LIN {X 0,Y 163.128,Z 425.869,A -85,B 0,C 180,E1 -26654.982,E2 -26654.982} C_VEL
LIN {X 0,Y 171.589,Z 416.887,A -85,B 0,C 180,E1 -26656.969,E2 -26656.969} C_VEL
LIN {X 0,Y 179.197,Z 407.097,A -85,B 0,C 180,E1 -26658.583,E2 -26658.583} C_VEL
LIN {X 0,Y 186.048,Z 396.461,A -85,B 0,C 180,E1 -26659.876,E2 -26659.876} C_VEL
LIN {X 0,Y 192.161,Z 384.861,A -85,B 0,C 180,E1 -26660.93,E2 -26660.93} C_VEL
LIN {X 0,Y 196.671,Z 373.993,A -85,B 0,C 180,E1 -26661.72,E2 -26661.72} C_VEL
LIN {X 0,Y 200.139,Z 363.217,A -85,B 0,C 180,E1 -26662.314,E2 -26662.314} C_VEL
LIN {X 0,Y 199.888,Z 363.628,A -85,B 0,C 180,E1 -26665.464,E2 -26665.464} C_VEL
LIN {X 0,Y 199.801,Z 364.596,A -85,B 0,C 180,E1 -26666.634,E2 -26666.634} C_VEL
LIN {X 0,Y 199.425,Z 366.277,A -85,B 0,C 180,E1 -26667.159,E2 -26667.159} C_VEL
LIN {X 0,Y 194.964,Z 379.043,A -85,B 0,C 180,E1 -26667.683,E2 -26667.683} C_VEL
LIN {X 0,Y 188.908,Z 392.245,A -85,B 0,C 180,E1 -26668.498,E2 -26668.498} C_VEL
LIN {X 0,Y 181.772,Z 404.47,A -85,B 0,C 180,E1 -26669.559,E2 -26669.559} C_VEL
LIN {X 0,Y 173.973,Z 415.421,A -85,B 0,C 180,E1 -26670.869,E2 -26670.869} C_VEL
LIN {X 0,Y 164.885,Z 425.886,A -85,B 0,C 180,E1 -26672.677,E2 -26672.677} C_VEL
LIN {X 0,Y 156.103,Z 434.387,A -85,B 0,C 180,E1 -26674.759,E2 -26674.759} C_VEL
LIN {X 0,Y 146.247,Z 442.42,A -85,B 0,C 180,E1 -26677.549,E2 -26677.549} C_VEL
LIN {X 0,Y 138.25,Z 447.941,A -85,B 0,C 180,E1 -26680.319,E2 -26680.319} C_VEL
LIN {X 0,Y 130.692,Z 452.389,A -85,B 0,C 180,E1 -26683.457,E2 -26683.457} C_VEL
LIN {X 0,Y 123.692,Z 455.88,A -85,B 0,C 180,E1 -26687.019,E2 -26687.019} C_VEL
LIN {X 0,Y 115.424,Z 459.143,A -85,B 0,C 180,E1 -26692.495,E2 -26692.495} C_VEL
LIN {X 0,Y 108.504,Z 460.97,A -85,B 0,C 180,E1 -26698.794,E2 -26698.794} C_VEL
LIN {X 0,Y 103.185,Z 461.402,A -85,B 0,C 180,E1 -26705.881,E2 -26705.881} C_VEL
LIN {X 0,Y 99.914,Z 460.389,A -85,B 0,C 180,E1 -26713.66,E2 -26713.66} C_VEL
LIN {X 0,Y 98.634,Z 457.962,A -85,B 0,C 180,E1 -26721.808,E2 -26721.808} C_VEL
LIN {X 0,Y 98.771,Z 454.798,A -85,B 0,C 180,E1 -26728.418,E2 -26728.418} C_VEL
LIN {X 0,Y 98.803,Z 451.965,A -85,B 0,C 180,E1 -26732.782,E2 -26732.782} C_VEL
LIN {X 0,Y 98.851,Z 447.513,A -85,B 0,C 180,E1 -26738.174,E2 -26738.174} C_VEL
LIN {X 0,Y 99.696,Z 441.144,A -85,B 0,C 180,E1 -26744.282,E2 -26744.282} C_VEL
LIN {X 0,Y 101.518,Z 433.131,A -85,B 0,C 180,E1 -26750.249,E2 -26750.249} C_VEL
LIN {X 0,Y 103.699,Z 424.917,A -85,B 0,C 180,E1 -26755.057,E2 -26755.057} C_VEL
LIN {X 0,Y 106.646,Z 414.958,A -85,B 0,C 180,E1 -26759.617,E2 -26759.617} C_VEL
LIN {X 0,Y 109.644,Z 404.598,A -85,B 0,C 180,E1 -26763.239,E2 -26763.239} C_VEL
LIN {X 0,Y 112.675,Z 392.942,A -85,B 0,C 180,E1 -26766.333,E2 -26766.333} C_VEL
LIN {X 0,Y 115.263,Z 381.156,A -85,B 0,C 180,E1 -26768.675,E2 -26768.675} C_VEL
LIN {X 0,Y 117.619,Z 367.853,A -85,B 0,C 180,E1 -26770.521,E2 -26770.521} C_VEL
LIN {X 0,Y 117.914,Z 365.846,A -85,B 0,C 180,E1 -26770.749,E2 -26770.749} C_VEL
LIN {X 0,Y 118.064,Z 360.135,A -85,B 0,C 180,E1 -26771.461,E2 -26771.461} C_VEL
LIN {X 0,Y 116.415,Z 350.753,A -85,B 0,C 180,E1 -26772.801,E2 -26772.801} C_VEL
LIN {X 0,Y 114.613,Z 341.305,A -85,B 0,C 180,E1 -26774.061,E2 -26774.061} C_VEL
LIN {X 0,Y 114.511,Z 335.482,A -85,B 0,C 180,E1 -26774.605,E2 -26774.605} C_VEL
LIN {X 0,Y 115.704,Z 319.854,A -85,B 0,C 180,E1 -26775.743,E2 -26775.743} C_VEL
LIN {X 0,Y 114.812,Z 307.519,A -85,B 0,C 180,E1 -26777.142,E2 -26777.142} C_VEL
LIN {X 0,Y 109.913,Z 291.288,A -85,B 0,C 180,E1 -26780.25,E2 -26780.25} C_VEL
LIN {X 0,Y 105.352,Z 279.17,A -85,B 0,C 180,E1 -26783.198,E2 -26783.198} C_VEL
LIN {X 0,Y 99.994,Z 269.239,A -85,B 0,C 180,E1 -26786.524,E2 -26786.524} C_VEL
LIN {X 0,Y 95.808,Z 262.103,A -85,B 0,C 180,E1 -26789.408,E2 -26789.408} C_VEL
LIN {X 0,Y 94.08,Z 259.671,A -85,B 0,C 180,E1 -26790.642,E2 -26790.642} C_VEL
LIN {X 0,Y 93.573,Z 257.823,A -85,B 0,C 180,E1 -26791.237,E2 -26791.237} C_VEL
LIN {X 0,Y 93.642,Z 257.821,A -85,B 0,C 180,E1 -26797.958,E2 -26797.958} C_VEL
LIN {X 0,Y 94.005,Z 257.76,A -85,B 0,C 180,E1 -26807.038,E2 -26807.038} C_VEL
LIN {X 0,Y 94.117,Z 257.761,A -85,B 0,C 180,E1 -26811.409,E2 -26811.409} C_VEL
LIN {X 0,Y 94.728,Z 257.639,A -85,B 0,C 180,E1 -26819.998,E2 -26819.998} C_VEL
LIN {X 0,Y 94.142,Z 257.758,A -85,B 0,C 180,E1 -26828.585,E2 -26828.585} C_VEL
LIN {X 0,Y 93.991,Z 257.751,A -85,B 0,C 180,E1 -26833.606,E2 -26833.606} C_VEL
LIN {X 0,Y 93.679,Z 257.773,A -85,B 0,C 180,E1 -26842.03,E2 -26842.03} C_VEL
LIN {X 0,Y 93.611,Z 257.818,A -85,B 0,C 180,E1 -26846.772,E2 -26846.772} C_VEL
LIN {X 0,Y 93.588,Z 257.807,A -85,B 0,C 180,E1 -26854.316,E2 -26854.316} C_VEL
LIN {X 0,Y 93.537,Z 257.792,A -85,B 0,C 180,E1 -26862.547,E2 -26862.547} C_VEL
LIN {X 0,Y 93.53,Z 257.835,A -85,B 0,C 180,E1 -26868.711,E2 -26868.711} C_VEL
LIN {X 0,Y 93.579,Z 257.793,A -85,B 0,C 180,E1 -26875.7,E2 -26875.7} C_VEL
LIN {X 0,Y 93.664,Z 257.819,A -85,B 0,C 180,E1 -26884.209,E2 -26884.209} C_VEL
LIN {X 0,Y 93.691,Z 257.806,A -85,B 0,C 180,E1 -26887.975,E2 -26887.975} C_VEL
LIN {X 0,Y 94.089,Z 257.765,A -85,B 0,C 180,E1 -26897.053,E2 -26897.053} C_VEL
LIN {X 0,Y 94.12,Z 257.747,A -85,B 0,C 180,E1 -26900.058,E2 -26900.058} C_VEL
LIN {X 0,Y 95.242,Z 260.722,A -85,B 0,C 180,E1 -26901.106,E2 -26901.106} C_VEL
LIN {X 0,Y 96.858,Z 262.736,A -85,B 0,C 180,E1 -26902.193,E2 -26902.193} C_VEL
LIN {X 0,Y 98.996,Z 266.163,A -85,B 0,C 180,E1 -26903.652,E2 -26903.652} C_VEL
LIN {X 0,Y 102.442,Z 271.693,A -85,B 0,C 180,E1 -26905.821,E2 -26905.821} C_VEL
LIN {X 0,Y 109.777,Z 287.544,A -85,B 0,C 180,E1 -26910.3,E2 -26910.3} C_VEL
LIN {X 0,Y 116.248,Z 304.133,A -85,B 0,C 180,E1 -26913.943,E2 -26913.943} C_VEL
LIN {X 0,Y 116.608,Z 305.841,A -85,B 0,C 180,E1 -26914.203,E2 -26914.203} C_VEL
LIN {X 0,Y 112.302,Z 350.785,A -85,B 0,C 180,E1 -26917.359,E2 -26917.359} C_VEL
LIN {X 0,Y 110.494,Z 363.82,A -85,B 0,C 180,E1 -26918.918,E2 -26918.918} C_VEL
LIN {X 0,Y 107.94,Z 377.265,A -85,B 0,C 180,E1 -26921.263,E2 -26921.263} C_VEL
LIN {X 0,Y 104.836,Z 389.887,A -85,B 0,C 180,E1 -26924.32,E2 -26924.32} C_VEL
LIN {X 0,Y 101.801,Z 401.041,A -85,B 0,C 180,E1 -26927.94,E2 -26927.94} C_VEL
LIN {X 0,Y 98.733,Z 411.262,A -85,B 0,C 180,E1 -26932.281,E2 -26932.281} C_VEL
LIN {X 0,Y 96.103,Z 419.877,A -85,B 0,C 180,E1 -26936.942,E2 -26936.942} C_VEL
LIN {X 0,Y 93.655,Z 428.33,A -85,B 0,C 180,E1 -26942.751,E2 -26942.751} C_VEL
LIN {X 0,Y 92.06,Z 435.208,A -85,B 0,C 180,E1 -26948.791,E2 -26948.791} C_VEL
LIN {X 0,Y 90.924,Z 441.541,A -85,B 0,C 180,E1 -26955.923,E2 -26955.923} C_VEL
LIN {X 0,Y 90.75,Z 445.601,A -85,B 0,C 180,E1 -26961.719,E2 -26961.719} C_VEL
LIN {X 0,Y 91.999,Z 450.233,A -85,B 0,C 180,E1 -26970.372,E2 -26970.372} C_VEL
LIN {X 0,Y 94.797,Z 453.146,A -85,B 0,C 180,E1 -26978.244,E2 -26978.244} C_VEL
LIN {X 0,Y 97.638,Z 454.379,A -85,B 0,C 180,E1 -26983.268,E2 -26983.268} C_VEL
LIN {X 0,Y 101.113,Z 454.988,A -85,B 0,C 180,E1 -26987.966,E2 -26987.966} C_VEL
LIN {X 0,Y 106.154,Z 454.979,A -85,B 0,C 180,E1 -26993.205,E2 -26993.205} C_VEL
LIN {X 0,Y 112.489,Z 454.028,A -85,B 0,C 180,E1 -26998.241,E2 -26998.241} C_VEL
LIN {X 0,Y 120.795,Z 451.707,A -85,B 0,C 180,E1 -27003.337,E2 -27003.337} C_VEL
LIN {X 0,Y 130.29,Z 447.868,A -85,B 0,C 180,E1 -27007.85,E2 -27007.85} C_VEL
LIN {X 0,Y 140.094,Z 442.584,A -85,B 0,C 180,E1 -27011.577,E2 -27011.577} C_VEL
LIN {X 0,Y 148.86,Z 436.826,A -85,B 0,C 180,E1 -27014.291,E2 -27014.291} C_VEL
LIN {X 0,Y 158.415,Z 429.249,A -85,B 0,C 180,E1 -27016.761,E2 -27016.761} C_VEL
LIN {X 0,Y 167.121,Z 420.854,A -85,B 0,C 180,E1 -27018.71,E2 -27018.71} C_VEL
LIN {X 0,Y 175.528,Z 411.15,A -85,B 0,C 180,E1 -27020.387,E2 -27020.387} C_VEL
LIN {X 0,Y 183.337,Z 400.242,A -85,B 0,C 180,E1 -27021.732,E2 -27021.732} C_VEL
LIN {X 0,Y 189.266,Z 390.03,A -85,B 0,C 180,E1 -27022.696,E2 -27022.696} C_VEL
LIN {X 0,Y 195.03,Z 377.557,A -85,B 0,C 180,E1 -27023.606,E2 -27023.606} C_VEL
LIN {X 0,Y 197.721,Z 370.368,A -85,B 0,C 180,E1 -27024.018,E2 -27024.018} C_VEL
LIN {X 0,Y 197.801,Z 370.092,A -85,B 0,C 180,E1 -27024.219,E2 -27024.219} C_VEL
LIN {X 0,Y 197.787,Z 370.277,A -85,B 0,C 180,E1 -27025.066,E2 -27025.066} C_VEL
LIN {X 0,Y 197.46,Z 371.297,A -85,B 0,C 180,E1 -27025.267,E2 -27025.267} C_VEL
LIN {X 0,Y 192.672,Z 383.338,A -85,B 0,C 180,E1 -27025.795,E2 -27025.795} C_VEL
LIN {X 0,Y 186.571,Z 395.367,A -85,B 0,C 180,E1 -27026.549,E2 -27026.549} C_VEL
LIN {X 0,Y 179.278,Z 406.879,A -85,B 0,C 180,E1 -27027.521,E2 -27027.521} C_VEL
LIN {X 0,Y 172.115,Z 416.231,A -85,B 0,C 180,E1 -27028.62,E2 -27028.62} C_VEL
LIN {X 0,Y 162.783,Z 426.49,A -85,B 0,C 180,E1 -27030.301,E2 -27030.301} C_VEL
LIN {X 0,Y 153.733,Z 434.831,A -85,B 0,C 180,E1 -27032.259,E2 -27032.259} C_VEL
LIN {X 0,Y 144.941,Z 441.634,A -85,B 0,C 180,E1 -27034.491,E2 -27034.491} C_VEL
LIN {X 0,Y 133.814,Z 448.805,A -85,B 0,C 180,E1 -27038.026,E2 -27038.026} C_VEL
LIN {X 0,Y 125.938,Z 452.982,A -85,B 0,C 180,E1 -27041.124,E2 -27041.124} C_VEL
LIN {X 0,Y 118.613,Z 456.212,A -85,B 0,C 180,E1 -27044.688,E2 -27044.688} C_VEL
LIN {X 0,Y 109.877,Z 459.205,A -85,B 0,C 180,E1 -27050.241,E2 -27050.241} C_VEL
LIN {X 0,Y 102.489,Z 460.771,A -85,B 0,C 180,E1 -27056.734,E2 -27056.734} C_VEL
LIN {X 0,Y 96.746,Z 460.91,A -85,B 0,C 180,E1 -27064.162,E2 -27064.162} C_VEL
LIN {X 0,Y 93.117,Z 459.687,A -85,B 0,C 180,E1 -27072.43,E2 -27072.43} C_VEL
LIN {X 0,Y 91.655,Z 457.019,A -85,B 0,C 180,E1 -27081.179,E2 -27081.179} C_VEL
LIN {X 0,Y 91.753,Z 453.772,A -85,B 0,C 180,E1 -27088.145,E2 -27088.145} C_VEL
LIN {X 0,Y 91.795,Z 450.795,A -85,B 0,C 180,E1 -27092.821,E2 -27092.821} C_VEL
LIN {X 0,Y 91.961,Z 444.993,A -85,B 0,C 180,E1 -27099.9,E2 -27099.9} C_VEL
LIN {X 0,Y 93.125,Z 438.095,A -85,B 0,C 180,E1 -27106.438,E2 -27106.438} C_VEL
LIN {X 0,Y 95.385,Z 429.412,A -85,B 0,C 180,E1 -27112.754,E2 -27112.754} C_VEL
LIN {X 0,Y 97.953,Z 420.469,A -85,B 0,C 180,E1 -27117.795,E2 -27117.795} C_VEL
LIN {X 0,Y 100.887,Z 410.694,A -85,B 0,C 180,E1 -27122.08,E2 -27122.08} C_VEL
LIN {X 0,Y 104.043,Z 399.823,A -85,B 0,C 180,E1 -27125.71,E2 -27125.71} C_VEL
LIN {X 0,Y 107.046,Z 388.339,A -85,B 0,C 180,E1 -27128.582,E2 -27128.582} C_VEL
LIN {X 0,Y 109.87,Z 375.3,A -85,B 0,C 180,E1 -27130.963,E2 -27130.963} C_VEL
LIN {X 0,Y 112.097,Z 361.245,A -85,B 0,C 180,E1 -27132.673,E2 -27132.673} C_VEL
LIN {X 0,Y 114.511,Z 335.482,A -85,B 0,C 180,E1 -27134.605,E2 -27134.605} C_VEL
LIN {X 0,Y 114.425,Z 329.67,A -85,B 0,C 180,E1 -27135.168,E2 -27135.168} C_VEL
LIN {X 0,Y 113.409,Z 324.025,A -85,B 0,C 180,E1 -27135.972,E2 -27135.972} C_VEL
LIN {X 0,Y 107.787,Z 305.825,A -85,B 0,C 180,E1 -27139.468,E2 -27139.468} C_VEL
LIN {X 0,Y 102.649,Z 289.521,A -85,B 0,C 180,E1 -27143.091,E2 -27143.091} C_VEL
LIN {X 0,Y 99.916,Z 282.46,A -85,B 0,C 180,E1 -27144.99,E2 -27144.99} C_VEL
LIN {X 0,Y 94.449,Z 272.371,A -85,B 0,C 180,E1 -27148.763,E2 -27148.763} C_VEL
LIN {X 0,Y 91.1,Z 266.722,A -85,B 0,C 180,E1 -27151.329,E2 -27151.329} C_VEL
LIN {X 0,Y 88.937,Z 263.157,A -85,B 0,C 180,E1 -27153.096,E2 -27153.096} C_VEL
LIN {X 0,Y 87.203,Z 260.823,A -85,B 0,C 180,E1 -27154.514,E2 -27154.514} C_VEL
LIN {X 0,Y 86.551,Z 258.691,A -85,B 0,C 180,E1 -27155.324,E2 -27155.324} C_VEL
LIN {X 0,Y 86.586,Z 258.685,A -85,B 0,C 180,E1 -27161.053,E2 -27161.053} C_VEL
LIN {X 0,Y 86.848,Z 258.643,A -85,B 0,C 180,E1 -27166.157,E2 -27166.157} C_VEL
LIN {X 0,Y 87.012,Z 258.647,A -85,B 0,C 180,E1 -27170.702,E2 -27170.702} C_VEL
LIN {X 0,Y 87.66,Z 258.517,A -85,B 0,C 180,E1 -27179.998,E2 -27179.998} C_VEL
LIN {X 0,Y 87.052,Z 258.64,A -85,B 0,C 180,E1 -27189.29,E2 -27189.29} C_VEL
LIN {X 0,Y 86.884,Z 258.629,A -85,B 0,C 180,E1 -27194.042,E2 -27194.042} C_VEL
LIN {X 0,Y 86.617,Z 258.63,A -85,B 0,C 180,E1 -27198.937,E2 -27198.937} C_VEL
LIN {X 0,Y 86.574,Z 258.695,A -85,B 0,C 180,E1 -27206.764,E2 -27206.764} C_VEL
LIN {X 0,Y 86.509,Z 258.673,A -85,B 0,C 180,E1 -27215.679,E2 -27215.679} C_VEL
LIN {X 0,Y 86.478,Z 258.673,A -85,B 0,C 180,E1 -27223.001,E2 -27223.001} C_VEL
LIN {X 0,Y 86.451,Z 258.717,A -85,B 0,C 180,E1 -27229.437,E2 -27229.437} C_VEL
LIN {X 0,Y 86.522,Z 258.673,A -85,B 0,C 180,E1 -27235.353,E2 -27235.353} C_VEL
LIN {X 0,Y 86.578,Z 258.697,A -85,B 0,C 180,E1 -27243.24,E2 -27243.24} C_VEL
LIN {X 0,Y 86.645,Z 258.667,A -85,B 0,C 180,E1 -27251.07,E2 -27251.07} C_VEL
LIN {X 0,Y 86.973,Z 258.822,A -85,B 0,C 180,E1 -27256.047,E2 -27256.047} C_VEL
LIN {X 0,Y 88.098,Z 261.576,A -85,B 0,C 180,E1 -27257.182,E2 -27257.182} C_VEL
LIN {X 0,Y 89.958,Z 263.827,A -85,B 0,C 180,E1 -27258.627,E2 -27258.627} C_VEL
LIN {X 0,Y 92.146,Z 267.211,A -85,B 0,C 180,E1 -27260.313,E2 -27260.313} C_VEL
LIN {X 0,Y 97.679,Z 276.274,A -85,B 0,C 180,E1 -27264.283,E2 -27264.283} C_VEL
LIN {X 0,Y 104.482,Z 291.419,A -85,B 0,C 180,E1 -27268.816,E2 -27268.816} C_VEL
LIN {X 0,Y 110.395,Z 306.934,A -85,B 0,C 180,E1 -27272.467,E2 -27272.467} C_VEL
LIN {X 0,Y 105.939,Z 351.171,A -85,B 0,C 180,E1 -27275.689,E2 -27275.689} C_VEL
LIN {X 0,Y 103.843,Z 365.269,A -85,B 0,C 180,E1 -27277.473,E2 -27277.473} C_VEL
LIN {X 0,Y 101.404,Z 377.429,A -85,B 0,C 180,E1 -27279.725,E2 -27279.725} C_VEL
LIN {X 0,Y 98.186,Z 390.026,A -85,B 0,C 180,E1 -27282.924,E2 -27282.924} C_VEL
LIN {X 0,Y 95.015,Z 401.091,A -85,B 0,C 180,E1 -27286.703,E2 -27286.703} C_VEL
LIN {X 0,Y 91.908,Z 410.953,A -85,B 0,C 180,E1 -27291.129,E2 -27291.129} C_VEL
LIN {X 0,Y 88.674,Z 421.047,A -85,B 0,C 180,E1 -27297.051,E2 -27297.051} C_VEL
LIN {X 0,Y 86.255,Z 429.325,A -85,B 0,C 180,E1 -27303.362,E2 -27303.362} C_VEL
LIN {X 0,Y 84.686,Z 436.002,A -85,B 0,C 180,E1 -27309.859,E2 -27309.859} C_VEL
LIN {X 0,Y 83.83,Z 441.309,A -85,B 0,C 180,E1 -27316.333,E2 -27316.333} C_VEL
LIN {X 0,Y 83.824,Z 446.332,A -85,B 0,C 180,E1 -27324.065,E2 -27324.065} C_VEL
LIN {X 0,Y 84.793,Z 449.444,A -85,B 0,C 180,E1 -27330.18,E2 -27330.18} C_VEL
LIN {X 0,Y 86.531,Z 451.862,A -85,B 0,C 180,E1 -27336.042,E2 -27336.042} C_VEL
LIN {X 0,Y 89.077,Z 453.627,A -85,B 0,C 180,E1 -27341.605,E2 -27341.605} C_VEL
LIN {X 0,Y 93.365,Z 455.008,A -85,B 0,C 180,E1 -27348.087,E2 -27348.087} C_VEL
LIN {X 0,Y 98.901,Z 455.475,A -85,B 0,C 180,E1 -27354.124,E2 -27354.124} C_VEL
LIN {X 0,Y 106.196,Z 454.869,A -85,B 0,C 180,E1 -27360.001,E2 -27360.001} C_VEL
LIN {X 0,Y 112.72,Z 453.53,A -85,B 0,C 180,E1 -27364.071,E2 -27364.071} C_VEL
LIN {X 0,Y 120.648,Z 451.105,A -85,B 0,C 180,E1 -27368.035,E2 -27368.035} C_VEL
LIN {X 0,Y 131.42,Z 446.582,A -85,B 0,C 180,E1 -27372.353,E2 -27372.353} C_VEL
LIN {X 0,Y 142.298,Z 440.543,A -85,B 0,C 180,E1 -27375.763,E2 -27375.763} C_VEL
LIN {X 0,Y 152.107,Z 433.74,A -85,B 0,C 180,E1 -27378.255,E2 -27378.255} C_VEL
LIN {X 0,Y 161.786,Z 425.663,A -85,B 0,C 180,E1 -27380.337,E2 -27380.337} C_VEL
LIN {X 0,Y 169.833,Z 417.552,A -85,B 0,C 180,E1 -27381.867,E2 -27381.867} C_VEL
LIN {X 0,Y 178.101,Z 407.515,A -85,B 0,C 180,E1 -27383.242,E2 -27383.242} C_VEL
LIN {X 0,Y 185.063,Z 397.262,A -85,B 0,C 180,E1 -27384.31,E2 -27384.31} C_VEL
LIN {X 0,Y 185.261,Z 396.969,A -85,B 0,C 180,E1 -27384.446,E2 -27384.446} C_VEL
LIN {X 0,Y 177.848,Z 408.08,A -85,B 0,C 180,E1 -27385.331,E2 -27385.331} C_VEL
LIN {X 0,Y 168.922,Z 419.053,A -85,B 0,C 180,E1 -27386.567,E2 -27386.567} C_VEL
LIN {X 0,Y 159.408,Z 428.609,A -85,B 0,C 180,E1 -27388.156,E2 -27388.156} C_VEL
LIN {X 0,Y 148.607,Z 437.623,A -85,B 0,C 180,E1 -27390.346,E2 -27390.346} C_VEL
LIN {X 0,Y 138.166,Z 444.759,A -85,B 0,C 180,E1 -27392.943,E2 -27392.943} C_VEL
LIN {X 0,Y 126.82,Z 451.066,A -85,B 0,C 180,E1 -27396.538,E2 -27396.538} C_VEL
LIN {X 0,Y 118.792,Z 454.631,A -85,B 0,C 180,E1 -27399.733,E2 -27399.733} C_VEL
LIN {X 0,Y 113.743,Z 456.55,A -85,B 0,C 180,E1 -27402.151,E2 -27402.151} C_VEL
LIN {X 0,Y 104.505,Z 459.218,A -85,B 0,C 180,E1 -27407.745,E2 -27407.745} C_VEL
LIN {X 0,Y 96.625,Z 460.493,A -85,B 0,C 180,E1 -27414.421,E2 -27414.421} C_VEL
LIN {X 0,Y 90.41,Z 460.407,A -85,B 0,C 180,E1 -27422.202,E2 -27422.202} C_VEL
LIN {X 0,Y 86.376,Z 458.929,A -85,B 0,C 180,E1 -27431.008,E2 -27431.008} C_VEL
LIN {X 0,Y 84.713,Z 455.996,A -85,B 0,C 180,E1 -27440.45,E2 -27440.45} C_VEL
LIN {X 0,Y 84.781,Z 452.603,A -85,B 0,C 180,E1 -27447.86,E2 -27447.86} C_VEL
LIN {X 0,Y 84.776,Z 449.419,A -85,B 0,C 180,E1 -27453.064,E2 -27453.064} C_VEL
LIN {X 0,Y 85.021,Z 443.356,A -85,B 0,C 180,E1 -27460.717,E2 -27460.717} C_VEL
LIN {X 0,Y 86.343,Z 436.124,A -85,B 0,C 180,E1 -27467.77,E2 -27467.77} C_VEL
LIN {X 0,Y 88.843,Z 427.113,A -85,B 0,C 180,E1 -27474.535,E2 -27474.535} C_VEL
LIN {X 0,Y 92.092,Z 416.683,A -85,B 0,C 180,E1 -27480.366,E2 -27480.366} C_VEL
LIN {X 0,Y 95.395,Z 406.131,A -85,B 0,C 180,E1 -27484.812,E2 -27484.812} C_VEL
LIN {X 0,Y 98.895,Z 394.05,A -85,B 0,C 180,E1 -27488.58,E2 -27488.58} C_VEL
LIN {X 0,Y 102.108,Z 381.146,A -85,B 0,C 180,E1 -27491.483,E2 -27491.483} C_VEL
LIN {X 0,Y 104.615,Z 368.197,A -85,B 0,C 180,E1 -27493.512,E2 -27493.512} C_VEL
LIN {X 0,Y 106.437,Z 354.841,A -85,B 0,C 180,E1 -27494.879,E2 -27494.879} C_VEL
LIN {X 0,Y 109.49,Z 320.718,A -85,B 0,C 180,E1 -27497.421,E2 -27497.421} C_VEL
LIN {X 0,Y 108.795,Z 309.728,A -85,B 0,C 180,E1 -27498.742,E2 -27498.742} C_VEL
LIN {X 0,Y 107.787,Z 305.825,A -85,B 0,C 180,E1 -27499.468,E2 -27499.468} C_VEL
LIN {X 0,Y 105.834,Z 300.741,A -85,B 0,C 180,E1 -27500.676,E2 -27500.676} C_VEL
LIN {X 0,Y 103.066,Z 296.263,A -85,B 0,C 180,E1 -27502.188,E2 -27502.188} C_VEL
LIN {X 0,Y 94.591,Z 285.371,A -85,B 0,C 180,E1 -27507.016,E2 -27507.016} C_VEL
LIN {X 0,Y 92.822,Z 282.379,A -85,B 0,C 180,E1 -27508.273,E2 -27508.273} C_VEL
LIN {X 0,Y 87.205,Z 272.194,A -85,B 0,C 180,E1 -27512.811,E2 -27512.811} C_VEL
LIN {X 0,Y 84.154,Z 267.566,A -85,B 0,C 180,E1 -27515.482,E2 -27515.482} C_VEL
LIN {X 0,Y 82.237,Z 264.377,A -85,B 0,C 180,E1 -27517.381,E2 -27517.381} C_VEL
LIN {X 0,Y 80.259,Z 262.081,A -85,B 0,C 180,E1 -27519.327,E2 -27519.327} C_VEL
LIN {X 0,Y 79.527,Z 259.567,A -85,B 0,C 180,E1 -27520.644,E2 -27520.644} C_VEL
LIN {X 0,Y 79.765,Z 259.521,A -85,B 0,C 180,E1 -27525.716,E2 -27525.716} C_VEL
LIN {X 0,Y 79.897,Z 259.532,A -85,B 0,C 180,E1 -27529.866,E2 -27529.866} C_VEL
LIN {X 0,Y 80.591,Z 259.396,A -85,B 0,C 180,E1 -27539.998,E2 -27539.998} C_VEL
LIN {X 0,Y 79.935,Z 259.523,A -85,B 0,C 180,E1 -27550.126,E2 -27550.126} C_VEL
LIN {X 0,Y 79.717,Z 259.504,A -85,B 0,C 180,E1 -27555.335,E2 -27555.335} C_VEL
LIN {X 0,Y 79.492,Z 259.522,A -85,B 0,C 180,E1 -27560.708,E2 -27560.708} C_VEL
LIN {X 0,Y 79.472,Z 259.583,A -85,B 0,C 180,E1 -27567.843,E2 -27567.843} C_VEL
LIN {X 0,Y 79.374,Z 259.59,A -85,B 0,C 180,E1 -27572.088,E2 -27572.088} C_VEL
LIN {X 0,Y 79.367,Z 259.539,A -85,B 0,C 180,E1 -27578.303,E2 -27578.303} C_VEL
LIN {X 0,Y 79.404,Z 259.574,A -85,B 0,C 180,E1 -27585.076,E2 -27585.076} C_VEL
LIN {X 0,Y 79.379,Z 259.583,A -85,B 0,C 180,E1 -27592.826,E2 -27592.826} C_VEL
LIN {X 0,Y 79.369,Z 259.555,A -85,B 0,C 180,E1 -27597.912,E2 -27597.912} C_VEL
LIN {X 0,Y 79.52,Z 259.578,A -85,B 0,C 180,E1 -27603.778,E2 -27603.778} C_VEL
LIN {X 0,Y 79.599,Z 259.729,A -85,B 0,C 180,E1 -27610.689,E2 -27610.689} C_VEL
LIN {X 0,Y 80.704,Z 262.533,A -85,B 0,C 180,E1 -27612.086,E2 -27612.086} C_VEL
LIN {X 0,Y 83.202,Z 265.112,A -85,B 0,C 180,E1 -27614.446,E2 -27614.446} C_VEL
LIN {X 0,Y 85.468,Z 268.513,A -85,B 0,C 180,E1 -27616.553,E2 -27616.553} C_VEL
LIN {X 0,Y 92.73,Z 280.259,A -85,B 0,C 180,E1 -27622.378,E2 -27622.378} C_VEL
LIN {X 0,Y 99.152,Z 295.087,A -85,B 0,C 180,E1 -27627.175,E2 -27627.175} C_VEL
LIN {X 0,Y 104.228,Z 308.469,A -85,B 0,C 180,E1 -27630.562,E2 -27630.562} C_VEL
LIN {X 0,Y 99.648,Z 351.758,A -85,B 0,C 180,E1 -27633.872,E2 -27633.872} C_VEL
LIN {X 0,Y 97.425,Z 365.715,A -85,B 0,C 180,E1 -27635.724,E2 -27635.724} C_VEL
LIN {X 0,Y 94.642,Z 378.579,A -85,B 0,C 180,E1 -27638.265,E2 -27638.265} C_VEL
LIN {X 0,Y 91.285,Z 390.948,A -85,B 0,C 180,E1 -27641.643,E2 -27641.643} C_VEL
LIN {X 0,Y 87.982,Z 401.823,A -85,B 0,C 180,E1 -27645.659,E2 -27645.659} C_VEL
LIN {X 0,Y 84.548,Z 412.241,A -85,B 0,C 180,E1 -27650.772,E2 -27650.772} C_VEL
LIN {X 0,Y 81.217,Z 422.183,A -85,B 0,C 180,E1 -27657.203,E2 -27657.203} C_VEL
LIN {X 0,Y 78.835,Z 430.291,A -85,B 0,C 180,E1 -27664.102,E2 -27664.102} C_VEL
LIN {X 0,Y 77.322,Z 436.817,A -85,B 0,C 180,E1 -27671.192,E2 -27671.192} C_VEL
LIN {X 0,Y 76.7,Z 441.235,A -85,B 0,C 180,E1 -27677.135,E2 -27677.135} C_VEL
LIN {X 0,Y 77.034,Z 446.961,A -85,B 0,C 180,E1 -27686.814,E2 -27686.814} C_VEL
LIN {X 0,Y 79.458,Z 451.306,A -85,B 0,C 180,E1 -27696.643,E2 -27696.643} C_VEL
LIN {X 0,Y 83.696,Z 454.109,A -85,B 0,C 180,E1 -27705.411,E2 -27705.411} C_VEL
LIN {X 0,Y 87.555,Z 455.237,A -85,B 0,C 180,E1 -27710.764,E2 -27710.764} C_VEL
LIN {X 0,Y 92.091,Z 455.805,A -85,B 0,C 180,E1 -27715.625,E2 -27715.625} C_VEL
LIN {X 0,Y 98.393,Z 455.724,A -85,B 0,C 180,E1 -27720.863,E2 -27720.863} C_VEL
LIN {X 0,Y 105.926,Z 454.727,A -85,B 0,C 180,E1 -27725.662,E2 -27725.662} C_VEL
LIN {X 0,Y 115.801,Z 452.303,A -85,B 0,C 180,E1 -27730.492,E2 -27730.492} C_VEL
LIN {X 0,Y 126.301,Z 448.477,A -85,B 0,C 180,E1 -27734.502,E2 -27734.502} C_VEL
LIN {X 0,Y 137.563,Z 442.928,A -85,B 0,C 180,E1 -27737.852,E2 -27737.852} C_VEL
LIN {X 0,Y 148.333,Z 436.272,A -85,B 0,C 180,E1 -27740.43,E2 -27740.43} C_VEL
LIN {X 0,Y 157.231,Z 429.516,A -85,B 0,C 180,E1 -27742.226,E2 -27742.226} C_VEL
LIN {X 0,Y 166.373,Z 421.141,A -85,B 0,C 180,E1 -27743.833,E2 -27743.833} C_VEL
LIN {X 0,Y 165.956,Z 421.632,A -85,B 0,C 180,E1 -27744.44,E2 -27744.44} C_VEL
LIN {X 0,Y 156.256,Z 430.695,A -85,B 0,C 180,E1 -27745.914,E2 -27745.914} C_VEL
LIN {X 0,Y 145.209,Z 439.14,A -85,B 0,C 180,E1 -27747.97,E2 -27747.97} C_VEL
LIN {X 0,Y 134.478,Z 445.863,A -85,B 0,C 180,E1 -27750.433,E2 -27750.433} C_VEL
LIN {X 0,Y 125.62,Z 450.454,A -85,B 0,C 180,E1 -27752.954,E2 -27752.954} C_VEL
LIN {X 0,Y 117.126,Z 454.063,A -85,B 0,C 180,E1 -27755.908,E2 -27755.908} C_VEL
LIN {X 0,Y 109.104,Z 456.792,A -85,B 0,C 180,E1 -27759.384,E2 -27759.384} C_VEL
LIN {X 0,Y 98.991,Z 459.262,A -85,B 0,C 180,E1 -27765.234,E2 -27765.234} C_VEL
LIN {X 0,Y 90.94,Z 460.209,A -85,B 0,C 180,E1 -27771.816,E2 -27771.816} C_VEL
LIN {X 0,Y 84.199,Z 459.826,A -85,B 0,C 180,E1 -27779.949,E2 -27779.949} C_VEL
LIN {X 0,Y 79.72,Z 458.085,A -85,B 0,C 180,E1 -27789.353,E2 -27789.353} C_VEL
LIN {X 0,Y 77.784,Z 454.951,A -85,B 0,C 180,E1 -27799.59,E2 -27799.59} C_VEL
LIN {X 0,Y 77.784,Z 451.568,A -85,B 0,C 180,E1 -27807.245,E2 -27807.245} C_VEL
LIN {X 0,Y 77.779,Z 449.051,A -85,B 0,C 180,E1 -27811.664,E2 -27811.664} C_VEL
LIN {X 0,Y 77.845,Z 443.86,A -85,B 0,C 180,E1 -27818.958,E2 -27818.958} C_VEL
LIN {X 0,Y 79.019,Z 436.749,A -85,B 0,C 180,E1 -27826.799,E2 -27826.799} C_VEL
LIN {X 0,Y 81.474,Z 427.975,A -85,B 0,C 180,E1 -27834.185,E2 -27834.185} C_VEL
LIN {X 0,Y 84.302,Z 418.926,A -85,B 0,C 180,E1 -27840.009,E2 -27840.009} C_VEL
LIN {X 0,Y 87.571,Z 408.991,A -85,B 0,C 180,E1 -27844.872,E2 -27844.872} C_VEL
LIN {X 0,Y 90.915,Z 398.496,A -85,B 0,C 180,E1 -27848.734,E2 -27848.734} C_VEL
LIN {X 0,Y 94.39,Z 386.225,A -85,B 0,C 180,E1 -27852.07,E2 -27852.07} C_VEL
LIN {X 0,Y 97.217,Z 373.942,A -85,B 0,C 180,E1 -27854.446,E2 -27854.446} C_VEL
LIN {X 0,Y 99.62,Z 359.76,A -85,B 0,C 180,E1 -27856.279,E2 -27856.279} C_VEL
LIN {X 0,Y 103.367,Z 321.146,A -85,B 0,C 180,E1 -27859.351,E2 -27859.351} C_VEL
LIN {X 0,Y 102.852,Z 311.765,A -85,B 0,C 180,E1 -27860.554,E2 -27860.554} C_VEL
LIN {X 0,Y 98.473,Z 296.576,A -85,B 0,C 180,E1 -27863.926,E2 -27863.926} C_VEL
LIN {X 0,Y 94.877,Z 286.554,A -85,B 0,C 180,E1 -27866.726,E2 -27866.726} C_VEL
LIN {X 0,Y 92.822,Z 282.379,A -85,B 0,C 180,E1 -27868.273,E2 -27868.273} C_VEL
LIN {X 0,Y 90.834,Z 279.827,A -85,B 0,C 180,E1 -27869.672,E2 -27869.672} C_VEL
LIN {X 0,Y 86.531,Z 277.148,A -85,B 0,C 180,E1 -27872.484,E2 -27872.484} C_VEL
LIN {X 0,Y 82.202,Z 274.75,A -85,B 0,C 180,E1 -27875.68,E2 -27875.68} C_VEL
LIN {X 0,Y 80.113,Z 272.58,A -85,B 0,C 180,E1 -27877.589,E2 -27877.589} C_VEL
LIN {X 0,Y 78.377,Z 269.787,A -85,B 0,C 180,E1 -27879.494,E2 -27879.494} C_VEL
LIN {X 0,Y 76.283,Z 266.816,A -85,B 0,C 180,E1 -27881.882,E2 -27881.882} C_VEL
LIN {X 0,Y 75.485,Z 265.352,A -85,B 0,C 180,E1 -27882.909,E2 -27882.909} C_VEL
LIN {X 0,Y 73.572,Z 263.048,A -85,B 0,C 180,E1 -27885.299,E2 -27885.299} C_VEL
LIN {X 0,Y 72.734,Z 260.403,A -85,B 0,C 180,E1 -27886.909,E2 -27886.909} C_VEL
LIN {X 0,Y 72.967,Z 260.374,A -85,B 0,C 180,E1 -27894.471,E2 -27894.471} C_VEL
LIN {X 0,Y 73.521,Z 260.275,A -85,B 0,C 180,E1 -27899.998,E2 -27899.998} C_VEL
LIN {X 0,Y 72.829,Z 260.402,A -85,B 0,C 180,E1 -27911.126,E2 -27911.126} C_VEL
LIN {X 0,Y 72.553,Z 260.382,A -85,B 0,C 180,E1 -27916.892,E2 -27916.892} C_VEL
LIN {X 0,Y 72.378,Z 260.424,A -85,B 0,C 180,E1 -27922.853,E2 -27922.853} C_VEL
LIN {X 0,Y 72.369,Z 260.47,A -85,B 0,C 180,E1 -27929.083,E2 -27929.083} C_VEL
LIN {X 0,Y 72.292,Z 260.437,A -85,B 0,C 180,E1 -27935.68,E2 -27935.68} C_VEL
LIN {X 0,Y 72.256,Z 260.437,A -85,B 0,C 180,E1 -27942.908,E2 -27942.908} C_VEL
LIN {X 0,Y 72.289,Z 260.476,A -85,B 0,C 180,E1 -27951.053,E2 -27951.053} C_VEL
LIN {X 0,Y 72.287,Z 260.45,A -85,B 0,C 180,E1 -27954.319,E2 -27954.319} C_VEL
LIN {X 0,Y 72.474,Z 260.582,A -85,B 0,C 180,E1 -27963.938,E2 -27963.938} C_VEL
LIN {X 0,Y 73.314,Z 263.163,A -85,B 0,C 180,E1 -27965.458,E2 -27965.458} C_VEL
LIN {X 0,Y 75.369,Z 265.376,A -85,B 0,C 180,E1 -27968.008,E2 -27968.008} C_VEL
LIN {X 0,Y 76.11,Z 266.158,A -85,B 0,C 180,E1 -27968.858,E2 -27968.858} C_VEL
LIN {X 0,Y 78.091,Z 269.255,A -85,B 0,C 180,E1 -27971.168,E2 -27971.168} C_VEL
LIN {X 0,Y 79.694,Z 271.053,A -85,B 0,C 180,E1 -27972.787,E2 -27972.787} C_VEL
LIN {X 0,Y 82.905,Z 276.186,A -85,B 0,C 180,E1 -27976.046,E2 -27976.046} C_VEL
LIN {X 0,Y 88.154,Z 285.042,A -85,B 0,C 180,E1 -27980.618,E2 -27980.618} C_VEL
LIN {X 0,Y 93.79,Z 298.436,A -85,B 0,C 180,E1 -27985.259,E2 -27985.259} C_VEL
LIN {X 0,Y 98.047,Z 309.988,A -85,B 0,C 180,E1 -27988.473,E2 -27988.473} C_VEL
LIN {X 0,Y 93.542,Z 351.214,A -85,B 0,C 180,E1 -27991.729,E2 -27991.729} C_VEL
LIN {X 0,Y 91.299,Z 365.007,A -85,B 0,C 180,E1 -27993.595,E2 -27993.595} C_VEL
LIN {X 0,Y 88.66,Z 377.041,A -85,B 0,C 180,E1 -27995.972,E2 -27995.972} C_VEL
LIN {X 0,Y 85.043,Z 389.859,A -85,B 0,C 180,E1 -27999.513,E2 -27999.513} C_VEL
LIN {X 0,Y 81.584,Z 400.874,A -85,B 0,C 180,E1 -28003.702,E2 -28003.702} C_VEL
LIN {X 0,Y 77.898,Z 411.478,A -85,B 0,C 180,E1 -28009.086,E2 -28009.086} C_VEL
LIN {X 0,Y 74.706,Z 420.61,A -85,B 0,C 180,E1 -28015.259,E2 -28015.259} C_VEL
LIN {X 0,Y 72.008,Z 429.075,A -85,B 0,C 180,E1 -28022.789,E2 -28022.789} C_VEL
LIN {X 0,Y 70.542,Z 434.98,A -85,B 0,C 180,E1 -28029.46,E2 -28029.46} C_VEL
LIN {X 0,Y 69.663,Z 440.45,A -85,B 0,C 180,E1 -28037.083,E2 -28037.083} C_VEL
LIN {X 0,Y 69.95,Z 446.055,A -85,B 0,C 180,E1 -28046.957,E2 -28046.957} C_VEL
LIN {X 0,Y 72.304,Z 450.571,A -85,B 0,C 180,E1 -28057.122,E2 -28057.122} C_VEL
LIN {X 0,Y 75.075,Z 452.85,A -85,B 0,C 180,E1 -28063.692,E2 -28063.692} C_VEL
LIN {X 0,Y 78.742,Z 454.557,A -85,B 0,C 180,E1 -28069.719,E2 -28069.719} C_VEL
LIN {X 0,Y 84.483,Z 455.862,A -85,B 0,C 180,E1 -28076.516,E2 -28076.516} C_VEL
LIN {X 0,Y 91.439,Z 456.259,A -85,B 0,C 180,E1 -28082.466,E2 -28082.466} C_VEL
LIN {X 0,Y 100.292,Z 455.596,A -85,B 0,C 180,E1 -28088.058,E2 -28088.058} C_VEL
LIN {X 0,Y 107.623,Z 454.272,A -85,B 0,C 180,E1 -28091.642,E2 -28091.642} C_VEL
LIN {X 0,Y 116.492,Z 451.877,A -85,B 0,C 180,E1 -28095.164,E2 -28095.164} C_VEL
LIN {X 0,Y 125.72,Z 448.521,A -85,B 0,C 180,E1 -28098.152,E2 -28098.152} C_VEL
LIN {X 0,Y 136.981,Z 443.179,A -85,B 0,C 180,E1 -28101.049,E2 -28101.049} C_VEL
LIN {X 0,Y 145.155,Z 438.376,A -85,B 0,C 180,E1 -28102.79,E2 -28102.79} C_VEL
LIN {X 0,Y 149.585,Z 435.415,A -85,B 0,C 180,E1 -28103.637,E2 -28103.637} C_VEL
LIN {X 0,Y 146.885,Z 437.409,A -85,B 0,C 180,E1 -28104.634,E2 -28104.634} C_VEL
LIN {X 0,Y 137.317,Z 443.508,A -85,B 0,C 180,E1 -28106.419,E2 -28106.419} C_VEL
LIN {X 0,Y 128.009,Z 448.458,A -85,B 0,C 180,E1 -28108.556,E2 -28108.556} C_VEL
LIN {X 0,Y 116.004,Z 453.507,A -85,B 0,C 180,E1 -28111.996,E2 -28111.996} C_VEL
LIN {X 0,Y 104.749,Z 457.046,A -85,B 0,C 180,E1 -28116.386,E2 -28116.386} C_VEL
LIN {X 0,Y 94.472,Z 459.108,A -85,B 0,C 180,E1 -28121.94,E2 -28121.94} C_VEL
LIN {X 0,Y 85.469,Z 459.819,A -85,B 0,C 180,E1 -28128.87,E2 -28128.87} C_VEL
LIN {X 0,Y 78.142,Z 459.194,A -85,B 0,C 180,E1 -28137.345,E2 -28137.345} C_VEL
LIN {X 0,Y 73.128,Z 457.224,A -85,B 0,C 180,E1 -28147.394,E2 -28147.394} C_VEL
LIN {X 0,Y 70.882,Z 453.765,A -85,B 0,C 180,E1 -28158.563,E2 -28158.563} C_VEL
LIN {X 0,Y 70.794,Z 450.396,A -85,B 0,C 180,E1 -28166.612,E2 -28166.612} C_VEL
LIN {X 0,Y 70.78,Z 447.56,A -85,B 0,C 180,E1 -28171.824,E2 -28171.824} C_VEL
LIN {X 0,Y 70.903,Z 442.128,A -85,B 0,C 180,E1 -28179.843,E2 -28179.843} C_VEL
LIN {X 0,Y 72.258,Z 434.657,A -85,B 0,C 180,E1 -28188.425,E2 -28188.425} C_VEL
LIN {X 0,Y 74.546,Z 427.17,A -85,B 0,C 180,E1 -28195.099,E2 -28195.099} C_VEL
LIN {X 0,Y 77.557,Z 418.03,A -85,B 0,C 180,E1 -28201.398,E2 -28201.398} C_VEL
LIN {X 0,Y 81.027,Z 407.934,A -85,B 0,C 180,E1 -28206.601,E2 -28206.601} C_VEL
LIN {X 0,Y 84.666,Z 396.914,A -85,B 0,C 180,E1 -28210.815,E2 -28210.815} C_VEL
LIN {X 0,Y 87.98,Z 385.77,A -85,B 0,C 180,E1 -28213.939,E2 -28213.939} C_VEL
LIN {X 0,Y 90.928,Z 373.453,A -85,B 0,C 180,E1 -28216.429,E2 -28216.429} C_VEL
LIN {X 0,Y 93.462,Z 359.181,A -85,B 0,C 180,E1 -28218.346,E2 -28218.346} C_VEL
LIN {X 0,Y 97.317,Z 321.938,A -85,B 0,C 180,E1 -28221.418,E2 -28221.418} C_VEL
LIN {X 0,Y 96.859,Z 313.411,A -85,B 0,C 180,E1 -28222.596,E2 -28222.596} C_VEL
LIN {X 0,Y 92.474,Z 297.965,A -85,B 0,C 180,E1 -28226.399,E2 -28226.399} C_VEL
LIN {X 0,Y 89.706,Z 290.047,A -85,B 0,C 180,E1 -28228.861,E2 -28228.861} C_VEL
LIN {X 0,Y 84.515,Z 279.844,A -85,B 0,C 180,E1 -28233.317,E2 -28233.317} C_VEL
LIN {X 0,Y 80.233,Z 272.76,A -85,B 0,C 180,E1 -28237.464,E2 -28237.464} C_VEL
LIN {X 0,Y 80.113,Z 272.58,A -85,B 0,C 180,E1 -28237.589,E2 -28237.589} C_VEL
LIN {X 0,Y 78.161,Z 270.5,A -85,B 0,C 180,E1 -28239.551,E2 -28239.551} C_VEL
LIN {X 0,Y 74.331,Z 268.585,A -85,B 0,C 180,E1 -28243.358,E2 -28243.358} C_VEL
LIN {X 0,Y 69.853,Z 266.963,A -85,B 0,C 180,E1 -28248.661,E2 -28248.661} C_VEL
LIN {X 0,Y 68.59,Z 266.13,A -85,B 0,C 180,E1 -28250.534,E2 -28250.534} C_VEL
LIN {X 0,Y 66.784,Z 263.979,A -85,B 0,C 180,E1 -28253.768,E2 -28253.768} C_VEL
LIN {X 0,Y 66.018,Z 261.219,A -85,B 0,C 180,E1 -28256.183,E2 -28256.183} C_VEL
LIN {X 0,Y 66.419,Z 261.158,A -85,B 0,C 180,E1 -28259.998,E2 -28259.998} C_VEL
LIN {X 0,Y 65.729,Z 261.274,A -85,B 0,C 180,E1 -28272.346,E2 -28272.346} C_VEL
LIN {X 0,Y 65.363,Z 261.272,A -85,B 0,C 180,E1 -28278.816,E2 -28278.816} C_VEL
LIN {X 0,Y 65.227,Z 261.341,A -85,B 0,C 180,E1 -28285.528,E2 -28285.528} C_VEL
LIN {X 0,Y 65.191,Z 261.351,A -85,B 0,C 180,E1 -28292.615,E2 -28292.615} C_VEL
LIN {X 0,Y 65.186,Z 261.303,A -85,B 0,C 180,E1 -28301.009,E2 -28301.009} C_VEL
LIN {X 0,Y 65.201,Z 261.363,A -85,B 0,C 180,E1 -28309.71,E2 -28309.71} C_VEL
LIN {X 0,Y 65.266,Z 261.522,A -85,B 0,C 180,E1 -28313.971,E2 -28313.971} C_VEL
LIN {X 0,Y 66.112,Z 264.074,A -85,B 0,C 180,E1 -28316.226,E2 -28316.226} C_VEL
LIN {X 0,Y 68.034,Z 266.148,A -85,B 0,C 180,E1 -28319.683,E2 -28319.683} C_VEL
LIN {X 0,Y 69.409,Z 267.143,A -85,B 0,C 180,E1 -28321.791,E2 -28321.791} C_VEL
LIN {X 0,Y 71.102,Z 270.204,A -85,B 0,C 180,E1 -28324.607,E2 -28324.607} C_VEL
LIN {X 0,Y 72.917,Z 272.249,A -85,B 0,C 180,E1 -28327.025,E2 -28327.025} C_VEL
LIN {X 0,Y 75.297,Z 275.637,A -85,B 0,C 180,E1 -28329.987,E2 -28329.987} C_VEL
LIN {X 0,Y 78.439,Z 280.486,A -85,B 0,C 180,E1 -28333.478,E2 -28333.478} C_VEL
LIN {X 0,Y 83.536,Z 289.438,A -85,B 0,C 180,E1 -28338.553,E2 -28338.553} C_VEL
LIN {X 0,Y 88.646,Z 302.139,A -85,B 0,C 180,E1 -28343.243,E2 -28343.243} C_VEL
LIN {X 0,Y 92.039,Z 311.971,A -85,B 0,C 180,E1 -28346.179,E2 -28346.179} C_VEL
LIN {X 0,Y 87.45,Z 351.706,A -85,B 0,C 180,E1 -28349.419,E2 -28349.419} C_VEL
LIN {X 0,Y 85.183,Z 364.871,A -85,B 0,C 180,E1 -28351.252,E2 -28351.252} C_VEL
LIN {X 0,Y 82.426,Z 376.848,A -85,B 0,C 180,E1 -28353.689,E2 -28353.689} C_VEL
LIN {X 0,Y 79.256,Z 387.799,A -85,B 0,C 180,E1 -28356.746,E2 -28356.746} C_VEL
LIN {X 0,Y 75.267,Z 399.858,A -85,B 0,C 180,E1 -28361.44,E2 -28361.44} C_VEL
LIN {X 0,Y 71.298,Z 410.697,A -85,B 0,C 180,E1 -28367.199,E2 -28367.199} C_VEL
LIN {X 0,Y 67.521,Z 420.828,A -85,B 0,C 180,E1 -28374.602,E2 -28374.602} C_VEL
LIN {X 0,Y 64.806,Z 429.218,A -85,B 0,C 180,E1 -28382.832,E2 -28382.832} C_VEL
LIN {X 0,Y 63.088,Z 436.347,A -85,B 0,C 180,E1 -28391.939,E2 -28391.939} C_VEL
LIN {X 0,Y 62.532,Z 442.409,A -85,B 0,C 180,E1 -28401.875,E2 -28401.875} C_VEL
LIN {X 0,Y 64.094,Z 448.123,A -85,B 0,C 180,E1 -28413.987,E2 -28413.987} C_VEL
LIN {X 0,Y 68.183,Z 452.29,A -85,B 0,C 180,E1 -28425.146,E2 -28425.146} C_VEL
LIN {X 0,Y 74.268,Z 455.003,A -85,B 0,C 180,E1 -28434.572,E2 -28434.572} C_VEL
LIN {X 0,Y 79.338,Z 456.069,A -85,B 0,C 180,E1 -28440.002,E2 -28440.002} C_VEL
LIN {X 0,Y 85.078,Z 456.615,A -85,B 0,C 180,E1 -28444.74,E2 -28444.74} C_VEL
LIN {X 0,Y 92.641,Z 456.498,A -85,B 0,C 180,E1 -28449.559,E2 -28449.559} C_VEL
LIN {X 0,Y 101.316,Z 455.502,A -85,B 0,C 180,E1 -28453.824,E2 -28453.824} C_VEL
LIN {X 0,Y 112.827,Z 452.992,A -85,B 0,C 180,E1 -28458.148,E2 -28458.148} C_VEL
LIN {X 0,Y 124.542,Z 449.073,A -85,B 0,C 180,E1 -28461.52,E2 -28461.52} C_VEL
LIN {X 0,Y 133.055,Z 445.354,A -85,B 0,C 180,E1 -28463.486,E2 -28463.486} C_VEL
LIN {X 0,Y 131.116,Z 446.364,A -85,B 0,C 180,E1 -28464.339,E2 -28464.339} C_VEL
LIN {X 0,Y 118.547,Z 451.907,A -85,B 0,C 180,E1 -28467.231,E2 -28467.231} C_VEL
LIN {X 0,Y 112.42,Z 454.044,A -85,B 0,C 180,E1 -28468.94,E2 -28468.94} C_VEL
LIN {X 0,Y 100.712,Z 457.186,A -85,B 0,C 180,E1 -28473.143,E2 -28473.143} C_VEL
LIN {X 0,Y 89.879,Z 458.971,A -85,B 0,C 180,E1 -28478.569,E2 -28478.569} C_VEL
LIN {X 0,Y 80.255,Z 459.422,A -85,B 0,C 180,E1 -28485.533,E2 -28485.533} C_VEL
LIN {X 0,Y 72.276,Z 458.496,A -85,B 0,C 180,E1 -28494.312,E2 -28494.312} C_VEL
LIN {X 0,Y 66.681,Z 456.233,A -85,B 0,C 180,E1 -28505.068,E2 -28505.068} C_VEL
LIN {X 0,Y 64.009,Z 452.569,A -85,B 0,C 180,E1 -28517.316,E2 -28517.316} C_VEL
LIN {X 0,Y 63.84,Z 449.153,A -85,B 0,C 180,E1 -28525.811,E2 -28525.811} C_VEL
LIN {X 0,Y 63.8,Z 445.932,A -85,B 0,C 180,E1 -28532.112,E2 -28532.112} C_VEL
LIN {X 0,Y 63.985,Z 440.252,A -85,B 0,C 180,E1 -28540.92,E2 -28540.92} C_VEL
LIN {X 0,Y 65.644,Z 432.451,A -85,B 0,C 180,E1 -28550.359,E2 -28550.359} C_VEL
LIN {X 0,Y 68.138,Z 424.567,A -85,B 0,C 180,E1 -28557.651,E2 -28557.651} C_VEL
LIN {X 0,Y 72.055,Z 413.946,A -85,B 0,C 180,E1 -28564.956,E2 -28564.956} C_VEL
LIN {X 0,Y 75.994,Z 402.999,A -85,B 0,C 180,E1 -28570.337,E2 -28570.337} C_VEL
LIN {X 0,Y 80.024,Z 390.783,A -85,B 0,C 180,E1 -28574.628,E2 -28574.628} C_VEL
LIN {X 0,Y 83.377,Z 378.804,A -85,B 0,C 180,E1 -28577.595,E2 -28577.595} C_VEL
LIN {X 0,Y 86.373,Z 364.898,A -85,B 0,C 180,E1 -28579.931,E2 -28579.931} C_VEL
LIN {X 0,Y 88.121,Z 352.797,A -85,B 0,C 180,E1 -28581.261,E2 -28581.261} C_VEL
LIN {X 0,Y 91.33,Z 322.191,A -85,B 0,C 180,E1 -28583.814,E2 -28583.814} C_VEL
LIN {X 0,Y 91.071,Z 315.433,A -85,B 0,C 180,E1 -28584.8,E2 -28584.8} C_VEL
LIN {X 0,Y 86.9,Z 300.096,A -85,B 0,C 180,E1 -28588.962,E2 -28588.962} C_VEL
LIN {X 0,Y 84.545,Z 293.482,A -85,B 0,C 180,E1 -28591.227,E2 -28591.227} C_VEL
LIN {X 0,Y 79.126,Z 282.487,A -85,B 0,C 180,E1 -28596.612,E2 -28596.612} C_VEL
LIN {X 0,Y 74.708,Z 275.213,A -85,B 0,C 180,E1 -28601.664,E2 -28601.664} C_VEL
LIN {X 0,Y 72.392,Z 271.502,A -85,B 0,C 180,E1 -28604.694,E2 -28604.694} C_VEL
LIN {X 0,Y 70.091,Z 268.176,A -85,B 0,C 180,E1 -28608.063,E2 -28608.063} C_VEL
LIN {X 0,Y 69.333,Z 266.614,A -85,B 0,C 180,E1 -28609.411,E2 -28609.411} C_VEL
LIN {X 0,Y 68.59,Z 266.13,A -85,B 0,C 180,E1 -28610.534,E2 -28610.534} C_VEL
LIN {X 0,Y 66.762,Z 265.303,A -85,B 0,C 180,E1 -28613.431,E2 -28613.431} C_VEL
LIN {X 0,Y 63.693,Z 265.596,A -85,B 0,C 180,E1 -28618.666,E2 -28618.666} C_VEL
LIN {X 0,Y 61.098,Z 266.039,A -85,B 0,C 180,E1 -28624.393,E2 -28624.393} C_VEL
LIN {X 0,Y 59.993,Z 265.428,A -85,B 0,C 180,E1 -28627.996,E2 -28627.996} C_VEL
LIN {X 0,Y 58.569,Z 262.674,A -85,B 0,C 180,E1 -28636.293,E2 -28636.293} C_VEL
LIN {X 0,Y 58.174,Z 262.173,A -85,B 0,C 180,E1 -28641.247,E2 -28641.247} C_VEL
LIN {X 0,Y 58.206,Z 262.416,A -85,B 0,C 180,E1 -28651.351,E2 -28651.351} C_VEL
LIN {X 0,Y 58.92,Z 264.811,A -85,B 0,C 180,E1 -28658.59,E2 -28658.59} C_VEL
LIN {X 0,Y 61.405,Z 267.411,A -85,B 0,C 180,E1 -28668.06,E2 -28668.06} C_VEL
LIN {X 0,Y 62.794,Z 268.193,A -85,B 0,C 180,E1 -28671.574,E2 -28671.574} C_VEL
LIN {X 0,Y 64.251,Z 271.165,A -85,B 0,C 180,E1 -28675.364,E2 -28675.364} C_VEL
LIN {X 0,Y 66.535,Z 273.315,A -85,B 0,C 180,E1 -28679.538,E2 -28679.538} C_VEL
LIN {X 0,Y 68.668,Z 276.756,A -85,B 0,C 180,E1 -28683.286,E2 -28683.286} C_VEL
LIN {X 0,Y 69.79,Z 278.283,A -85,B 0,C 180,E1 -28684.997,E2 -28684.997} C_VEL
LIN {X 0,Y 73.086,Z 283.128,A -85,B 0,C 180,E1 -28689.465,E2 -28689.465} C_VEL
LIN {X 0,Y 77.739,Z 291.34,A -85,B 0,C 180,E1 -28694.867,E2 -28694.867} C_VEL
LIN {X 0,Y 79.541,Z 295.246,A -85,B 0,C 180,E1 -28696.851,E2 -28696.851} C_VEL
LIN {X 0,Y 83.784,Z 306.498,A -85,B 0,C 180,E1 -28701.278,E2 -28701.278} C_VEL
LIN {X 0,Y 86.175,Z 313.517,A -85,B 0,C 180,E1 -28703.568,E2 -28703.568} C_VEL
LIN {X 0,Y 81.4,Z 352.285,A -85,B 0,C 180,E1 -28706.834,E2 -28706.834} C_VEL
LIN {X 0,Y 78.962,Z 365.589,A -85,B 0,C 180,E1 -28708.787,E2 -28708.787} C_VEL
LIN {X 0,Y 75.974,Z 377.704,A -85,B 0,C 180,E1 -28711.402,E2 -28711.402} C_VEL
LIN {X 0,Y 72.072,Z 390.118,A -85,B 0,C 180,E1 -28715.21,E2 -28715.21} C_VEL
LIN {X 0,Y 68.172,Z 401.054,A -85,B 0,C 180,E1 -28719.91,E2 -28719.91} C_VEL
LIN {X 0,Y 64.171,Z 411.348,A -85,B 0,C 180,E1 -28725.943,E2 -28725.943} C_VEL
LIN {X 0,Y 60.207,Z 421.452,A -85,B 0,C 180,E1 -28734.181,E2 -28734.181} C_VEL
LIN {X 0,Y 57.435,Z 429.931,A -85,B 0,C 180,E1 -28743.601,E2 -28743.601} C_VEL
LIN {X 0,Y 55.844,Z 436.671,A -85,B 0,C 180,E1 -28753.484,E2 -28753.484} C_VEL
LIN {X 0,Y 55.659,Z 443.007,A -85,B 0,C 180,E1 -28765.378,E2 -28765.378} C_VEL
LIN {X 0,Y 58.11,Z 448.648,A -85,B 0,C 180,E1 -28778.729,E2 -28778.729} C_VEL
LIN {X 0,Y 61.246,Z 451.559,A -85,B 0,C 180,E1 -28786.735,E2 -28786.735} C_VEL
LIN {X 0,Y 65.382,Z 453.756,A -85,B 0,C 180,E1 -28793.832,E2 -28793.832} C_VEL
LIN {X 0,Y 70.401,Z 455.42,A -85,B 0,C 180,E1 -28800.002,E2 -28800.002} C_VEL
LIN {X 0,Y 77.817,Z 456.685,A -85,B 0,C 180,E1 -28806.607,E2 -28806.607} C_VEL
LIN {X 0,Y 86.202,Z 457.05,A -85,B 0,C 180,E1 -28811.971,E2 -28811.971} C_VEL
LIN {X 0,Y 96.657,Z 456.365,A -85,B 0,C 180,E1 -28816.91,E2 -28816.91} C_VEL
LIN {X 0,Y 104.544,Z 455.105,A -85,B 0,C 180,E1 -28819.771,E2 -28819.771} C_VEL
LIN {X 0,Y 116.069,Z 452.236,A -85,B 0,C 180,E1 -28823.133,E2 -28823.133} C_VEL
LIN {X 0,Y 115.482,Z 452.508,A -85,B 0,C 180,E1 -28824.109,E2 -28824.109} C_VEL
LIN {X 0,Y 103.021,Z 456.082,A -85,B 0,C 180,E1 -28827.531,E2 -28827.531} C_VEL
LIN {X 0,Y 91.221,Z 458.223,A -85,B 0,C 180,E1 -28832.071,E2 -28832.071} C_VEL
LIN {X 0,Y 80.313,Z 459.004,A -85,B 0,C 180,E1 -28838.049,E2 -28838.049} C_VEL
LIN {X 0,Y 70.813,Z 458.488,A -85,B 0,C 180,E1 -28846,E2 -28846} C_VEL
LIN {X 0,Y 63.145,Z 456.654,A -85,B 0,C 180,E1 -28856.19,E2 -28856.19} C_VEL
LIN {X 0,Y 58.346,Z 453.411,A -85,B 0,C 180,E1 -28868.818,E2 -28868.818} C_VEL
LIN {X 0,Y 56.899,Z 448.659,A -85,B 0,C 180,E1 -28882.905,E2 -28882.905} C_VEL
LIN {X 0,Y 56.89,Z 445.512,A -85,B 0,C 180,E1 -28889.999,E2 -28889.999} C_VEL
LIN {X 0,Y 56.937,Z 439.58,A -85,B 0,C 180,E1 -28900.309,E2 -28900.309} C_VEL
LIN {X 0,Y 58.643,Z 431.532,A -85,B 0,C 180,E1 -28911.068,E2 -28911.068} C_VEL
LIN {X 0,Y 61.326,Z 423.548,A -85,B 0,C 180,E1 -28919.143,E2 -28919.143} C_VEL
LIN {X 0,Y 65.076,Z 413.841,A -85,B 0,C 180,E1 -28926.435,E2 -28926.435} C_VEL
LIN {X 0,Y 69.254,Z 403.06,A -85,B 0,C 180,E1 -28932.24,E2 -28932.24} C_VEL
LIN {X 0,Y 73.495,Z 391.013,A -85,B 0,C 180,E1 -28936.807,E2 -28936.807} C_VEL
LIN {X 0,Y 77.177,Z 378.735,A -85,B 0,C 180,E1 -28940.047,E2 -28940.047} C_VEL
LIN {X 0,Y 80.273,Z 365.178,A -85,B 0,C 180,E1 -28942.452,E2 -28942.452} C_VEL
LIN {X 0,Y 82.222,Z 352.619,A -85,B 0,C 180,E1 -28943.903,E2 -28943.903} C_VEL
LIN {X 0,Y 85.573,Z 322.286,A -85,B 0,C 180,E1 -28946.538,E2 -28946.538} C_VEL
LIN {X 0,Y 85.42,Z 317.488,A -85,B 0,C 180,E1 -28947.288,E2 -28947.288} C_VEL
LIN {X 0,Y 81.678,Z 303.167,A -85,B 0,C 180,E1 -28951.473,E2 -28951.473} C_VEL
LIN {X 0,Y 79.369,Z 296.463,A -85,B 0,C 180,E1 -28954.05,E2 -28954.05} C_VEL
LIN {X 0,Y 74.634,Z 286.668,A -85,B 0,C 180,E1 -28959.5,E2 -28959.5} C_VEL
LIN {X 0,Y 71.105,Z 280.589,A -85,B 0,C 180,E1 -28964.042,E2 -28964.042} C_VEL
LIN {X 0,Y 68.215,Z 275.891,A -85,B 0,C 180,E1 -28968.483,E2 -28968.483} C_VEL
LIN {X 0,Y 66.319,Z 272.602,A -85,B 0,C 180,E1 -28972.003,E2 -28972.003} C_VEL
LIN {X 0,Y 64.222,Z 270.093,A -85,B 0,C 180,E1 -28976.078,E2 -28976.078} C_VEL
LIN {X 0,Y 63.26,Z 267.619,A -85,B 0,C 180,E1 -28978.708,E2 -28978.708} C_VEL
LIN {X 0,Y 59.993,Z 265.428,A -85,B 0,C 180,E1 -28987.996,E2 -28987.996} C_VEL
LIN {X 0,Y 59.143,Z 264.783,A -85,B 0,C 180,E1 -28991.601,E2 -28991.601} C_VEL
LIN {X 0,Y 58.365,Z 264.943,A -85,B 0,C 180,E1 -28995.341,E2 -28995.341} C_VEL
LIN {X 0,Y 57.464,Z 266.227,A -85,B 0,C 180,E1 -29001.034,E2 -29001.034} C_VEL
LIN {X 0,Y 57.161,Z 270.979,A -85,B 0,C 180,E1 -29014.669,E2 -29014.669} C_VEL
LIN {X 0,Y 57.715,Z 271.924,A -85,B 0,C 180,E1 -29018.639,E2 -29018.639} C_VEL
LIN {X 0,Y 59.59,Z 274.106,A -85,B 0,C 180,E1 -29026.362,E2 -29026.362} C_VEL
LIN {X 0,Y 60.612,Z 274.814,A -85,B 0,C 180,E1 -29029.38,E2 -29029.38} C_VEL
LIN {X 0,Y 62.461,Z 278.15,A -85,B 0,C 180,E1 -29034.519,E2 -29034.519} C_VEL
LIN {X 0,Y 63.957,Z 279.829,A -85,B 0,C 180,E1 -29037.597,E2 -29037.597} C_VEL
LIN {X 0,Y 67.105,Z 284.757,A -85,B 0,C 180,E1 -29043.347,E2 -29043.347} C_VEL
LIN {X 0,Y 70.091,Z 289.387,A -85,B 0,C 180,E1 -29047.85,E2 -29047.85} C_VEL
LIN {X 0,Y 74.717,Z 298.598,A -85,B 0,C 180,E1 -29053.838,E2 -29053.838} C_VEL
LIN {X 0,Y 78.742,Z 309.963,A -85,B 0,C 180,E1 -29058.74,E2 -29058.74} C_VEL
LIN {X 0,Y 80.421,Z 315.282,A -85,B 0,C 180,E1 -29060.648,E2 -29060.648} C_VEL
LIN {X 0,Y 75.585,Z 352.594,A -85,B 0,C 180,E1 -29063.857,E2 -29063.857} C_VEL
LIN {X 0,Y 73.029,Z 365.763,A -85,B 0,C 180,E1 -29065.835,E2 -29065.835} C_VEL
LIN {X 0,Y 69.907,Z 377.759,A -85,B 0,C 180,E1 -29068.505,E2 -29068.505} C_VEL
LIN {X 0,Y 65.586,Z 390.746,A -85,B 0,C 180,E1 -29072.687,E2 -29072.687} C_VEL
LIN {X 0,Y 61.651,Z 401,A -85,B 0,C 180,E1 -29077.368,E2 -29077.368} C_VEL
LIN {X 0,Y 57.179,Z 411.765,A -85,B 0,C 180,E1 -29084.229,E2 -29084.229} C_VEL
LIN {X 0,Y 52.943,Z 421.826,A -85,B 0,C 180,E1 -29093.466,E2 -29093.466} C_VEL
LIN {X 0,Y 50.127,Z 430.171,A -85,B 0,C 180,E1 -29104.109,E2 -29104.109} C_VEL
LIN {X 0,Y 48.615,Z 437.346,A -85,B 0,C 180,E1 -29116.283,E2 -29116.283} C_VEL
LIN {X 0,Y 48.966,Z 443.415,A -85,B 0,C 180,E1 -29129.438,E2 -29129.438} C_VEL
LIN {X 0,Y 52.574,Z 449.133,A -85,B 0,C 180,E1 -29144.496,E2 -29144.496} C_VEL
LIN {X 0,Y 58.949,Z 453.176,A -85,B 0,C 180,E1 -29156.656,E2 -29156.656} C_VEL
LIN {X 0,Y 67.235,Z 455.831,A -85,B 0,C 180,E1 -29166.002,E2 -29166.002} C_VEL
LIN {X 0,Y 73.647,Z 456.877,A -85,B 0,C 180,E1 -29171.005,E2 -29171.005} C_VEL
LIN {X 0,Y 80.648,Z 457.416,A -85,B 0,C 180,E1 -29175.157,E2 -29175.157} C_VEL
LIN {X 0,Y 89.247,Z 457.3,A -85,B 0,C 180,E1 -29179.112,E2 -29179.112} C_VEL
LIN {X 0,Y 98.886,Z 456.347,A -85,B 0,C 180,E1 -29182.507,E2 -29182.507} C_VEL
LIN {X 0,Y 99.939,Z 456.282,A -85,B 0,C 180,E1 -29183.921,E2 -29183.921} C_VEL
LIN {X 0,Y 87.656,Z 458.101,A -85,B 0,C 180,E1 -29188.133,E2 -29188.133} C_VEL
LIN {X 0,Y 76.134,Z 458.608,A -85,B 0,C 180,E1 -29193.828,E2 -29193.828} C_VEL
LIN {X 0,Y 65.898,Z 457.811,A -85,B 0,C 180,E1 -29201.715,E2 -29201.715} C_VEL
LIN {X 0,Y 57.425,Z 455.656,A -85,B 0,C 180,E1 -29212.275,E2 -29212.275} C_VEL
LIN {X 0,Y 51.881,Z 452.159,A -85,B 0,C 180,E1 -29226.024,E2 -29226.024} C_VEL
LIN {X 0,Y 50.04,Z 447.124,A -85,B 0,C 180,E1 -29241.926,E2 -29241.926} C_VEL
LIN {X 0,Y 49.928,Z 443.759,A -85,B 0,C 180,E1 -29249.999,E2 -29249.999} C_VEL
LIN {X 0,Y 50.057,Z 437.528,A -85,B 0,C 180,E1 -29261.744,E2 -29261.744} C_VEL
LIN {X 0,Y 52.151,Z 429.152,A -85,B 0,C 180,E1 -29273.843,E2 -29273.843} C_VEL
LIN {X 0,Y 55.281,Z 420.731,A -85,B 0,C 180,E1 -29282.7,E2 -29282.7} C_VEL
LIN {X 0,Y 59.604,Z 410.427,A -85,B 0,C 180,E1 -29290.423,E2 -29290.423} C_VEL
LIN {X 0,Y 64.232,Z 398.907,A -85,B 0,C 180,E1 -29296.451,E2 -29296.451} C_VEL
LIN {X 0,Y 68.308,Z 387.598,A -85,B 0,C 180,E1 -29300.494,E2 -29300.494} C_VEL
LIN {X 0,Y 71.807,Z 375.836,A -85,B 0,C 180,E1 -29303.456,E2 -29303.456} C_VEL
LIN {X 0,Y 74.9,Z 362.529,A -85,B 0,C 180,E1 -29305.694,E2 -29305.694} C_VEL
LIN {X 0,Y 77.064,Z 347.014,A -85,B 0,C 180,E1 -29307.349,E2 -29307.349} C_VEL
LIN {X 0,Y 79.891,Z 322.836,A -85,B 0,C 180,E1 -29309.493,E2 -29309.493} C_VEL
LIN {X 0,Y 79.742,Z 318.925,A -85,B 0,C 180,E1 -29310.192,E2 -29310.192} C_VEL
LIN {X 0,Y 76.438,Z 305.561,A -85,B 0,C 180,E1 -29314.582,E2 -29314.582} C_VEL
LIN {X 0,Y 74.756,Z 300.423,A -85,B 0,C 180,E1 -29316.799,E2 -29316.799} C_VEL
LIN {X 0,Y 70.458,Z 291.174,A -85,B 0,C 180,E1 -29322.399,E2 -29322.399} C_VEL
LIN {X 0,Y 67.431,Z 285.596,A -85,B 0,C 180,E1 -29327.01,E2 -29327.01} C_VEL
LIN {X 0,Y 64.919,Z 281.128,A -85,B 0,C 180,E1 -29331.633,E2 -29331.633} C_VEL
LIN {X 0,Y 63.537,Z 278.631,A -85,B 0,C 180,E1 -29334.502,E2 -29334.502} C_VEL
LIN {X 0,Y 61.485,Z 275.603,A -85,B 0,C 180,E1 -29339.334,E2 -29339.334} C_VEL
LIN {X 0,Y 60.907,Z 274.032,A -85,B 0,C 180,E1 -29341.237,E2 -29341.237} C_VEL
LIN {X 0,Y 58.054,Z 271.639,A -85,B 0,C 180,E1 -29351.211,E2 -29351.211} C_VEL
LIN {X 0,Y 57.192,Z 269.454,A -85,B 0,C 180,E1 -29357.984,E2 -29357.984} C_VEL
LIN {X 0,Y 56.913,Z 269.167,A -85,B 0,C 180,E1 -29361.741,E2 -29361.741} C_VEL
LIN {X 0,Y 56.948,Z 269.3,A -85,B 0,C 180,E1 -29369.907,E2 -29369.907} C_VEL
LIN {X 0,Y 57.471,Z 271.608,A -85,B 0,C 180,E1 -29377.186,E2 -29377.186} C_VEL
LIN {X 0,Y 57.715,Z 271.924,A -85,B 0,C 180,E1 -29378.639,E2 -29378.639} C_VEL
LIN {X 0,Y 58.444,Z 273.064,A -85,B 0,C 180,E1 -29382.255,E2 -29382.255} C_VEL
LIN {X 0,Y 59.166,Z 274.933,A -85,B 0,C 180,E1 -29385.542,E2 -29385.542} C_VEL
LIN {X 0,Y 60.516,Z 279.989,A -85,B 0,C 180,E1 -29391.283,E2 -29391.283} C_VEL
LIN {X 0,Y 63.184,Z 288.729,A -85,B 0,C 180,E1 -29399.058,E2 -29399.058} C_VEL
LIN {X 0,Y 64.526,Z 291.304,A -85,B 0,C 180,E1 -29401.681,E2 -29401.681} C_VEL
LIN {X 0,Y 66.635,Z 294.895,A -85,B 0,C 180,E1 -29405.308,E2 -29405.308} C_VEL
LIN {X 0,Y 70.339,Z 302.853,A -85,B 0,C 180,E1 -29410.951,E2 -29410.951} C_VEL
LIN {X 0,Y 73.907,Z 313.559,A -85,B 0,C 180,E1 -29415.932,E2 -29415.932} C_VEL
LIN {X 0,Y 74.917,Z 317.003,A -85,B 0,C 180,E1 -29417.294,E2 -29417.294} C_VEL
LIN {X 0,Y 69.994,Z 352.985,A -85,B 0,C 180,E1 -29420.417,E2 -29420.417} C_VEL
LIN {X 0,Y 67.345,Z 365.747,A -85,B 0,C 180,E1 -29422.355,E2 -29422.355} C_VEL
LIN {X 0,Y 63.94,Z 378.012,A -85,B 0,C 180,E1 -29425.154,E2 -29425.154} C_VEL
LIN {X 0,Y 59.502,Z 390.543,A -85,B 0,C 180,E1 -29429.35,E2 -29429.35} C_VEL
LIN {X 0,Y 54.756,Z 401.978,A -85,B 0,C 180,E1 -29434.957,E2 -29434.957} C_VEL
LIN {X 0,Y 49.987,Z 412.645,A -85,B 0,C 180,E1 -29442.619,E2 -29442.619} C_VEL
LIN {X 0,Y 45.681,Z 422.192,A -85,B 0,C 180,E1 -29452.625,E2 -29452.625} C_VEL
LIN {X 0,Y 42.833,Z 430.455,A -85,B 0,C 180,E1 -29464.882,E2 -29464.882} C_VEL
LIN {X 0,Y 41.527,Z 436.804,A -85,B 0,C 180,E1 -29477.398,E2 -29477.398} C_VEL
LIN {X 0,Y 42.314,Z 443.037,A -85,B 0,C 180,E1 -29492.826,E2 -29492.826} C_VEL
LIN {X 0,Y 45.872,Z 448.083,A -85,B 0,C 180,E1 -29507.075,E2 -29507.075} C_VEL
LIN {X 0,Y 52.58,Z 452.415,A -85,B 0,C 180,E1 -29520.003,E2 -29520.003} C_VEL
LIN {X 0,Y 58.382,Z 454.581,A -85,B 0,C 180,E1 -29526.917,E2 -29526.917} C_VEL
LIN {X 0,Y 64.876,Z 456.219,A -85,B 0,C 180,E1 -29532.515,E2 -29532.515} C_VEL
LIN {X 0,Y 73.929,Z 457.475,A -85,B 0,C 180,E1 -29538.096,E2 -29538.096} C_VEL
LIN {X 0,Y 83.571,Z 457.848,A -85,B 0,C 180,E1 -29542.337,E2 -29542.337} C_VEL
LIN {X 0,Y 84.546,Z 457.938,A -85,B 0,C 180,E1 -29543.895,E2 -29543.895} C_VEL
LIN {X 0,Y 72.418,Z 458.107,A -85,B 0,C 180,E1 -29549.151,E2 -29549.151} C_VEL
LIN {X 0,Y 61.411,Z 457.022,A -85,B 0,C 180,E1 -29556.773,E2 -29556.773} C_VEL
LIN {X 0,Y 52.031,Z 454.613,A -85,B 0,C 180,E1 -29567.522,E2 -29567.522} C_VEL
LIN {X 0,Y 45.575,Z 450.817,A -85,B 0,C 180,E1 -29582.446,E2 -29582.446} C_VEL
LIN {X 0,Y 43.323,Z 446.742,A -85,B 0,C 180,E1 -29596.755,E2 -29596.755} C_VEL
LIN {X 0,Y 43.128,Z 443.817,A -85,B 0,C 180,E1 -29605.326,E2 -29605.326} C_VEL
LIN {X 0,Y 42.864,Z 440.415,A -85,B 0,C 180,E1 -29613.411,E2 -29613.411} C_VEL
LIN {X 0,Y 43.524,Z 433.909,A -85,B 0,C 180,E1 -29626.171,E2 -29626.171} C_VEL
LIN {X 0,Y 46.48,Z 424.883,A -85,B 0,C 180,E1 -29639.429,E2 -29639.429} C_VEL
LIN {X 0,Y 50.906,Z 414.616,A -85,B 0,C 180,E1 -29649.676,E2 -29649.676} C_VEL
LIN {X 0,Y 55.52,Z 404.258,A -85,B 0,C 180,E1 -29656.7,E2 -29656.7} C_VEL
LIN {X 0,Y 60.239,Z 392.801,A -85,B 0,C 180,E1 -29661.944,E2 -29661.944} C_VEL
LIN {X 0,Y 64.756,Z 379.876,A -85,B 0,C 180,E1 -29665.837,E2 -29665.837} C_VEL
LIN {X 0,Y 68.262,Z 366.674,A -85,B 0,C 180,E1 -29668.481,E2 -29668.481} C_VEL
LIN {X 0,Y 70.652,Z 353.847,A -85,B 0,C 180,E1 -29670.1,E2 -29670.1} C_VEL
LIN {X 0,Y 74.464,Z 323.565,A -85,B 0,C 180,E1 -29672.851,E2 -29672.851} C_VEL
LIN {X 0,Y 74.29,Z 320.496,A -85,B 0,C 180,E1 -29673.517,E2 -29673.517} C_VEL
LIN {X 0,Y 71.355,Z 307.717,A -85,B 0,C 180,E1 -29678.212,E2 -29678.212} C_VEL
LIN {X 0,Y 69.228,Z 301.921,A -85,B 0,C 180,E1 -29681.309,E2 -29681.309} C_VEL
LIN {X 0,Y 66.002,Z 294.504,A -85,B 0,C 180,E1 -29686.528,E2 -29686.528} C_VEL
LIN {X 0,Y 62.487,Z 287.605,A -85,B 0,C 180,E1 -29693.407,E2 -29693.407} C_VEL
LIN {X 0,Y 60.843,Z 284.614,A -85,B 0,C 180,E1 -29697.272,E2 -29697.272} C_VEL
LIN {X 0,Y 58.941,Z 281.002,A -85,B 0,C 180,E1 -29702.988,E2 -29702.988} C_VEL
LIN {X 0,Y 58.023,Z 280.119,A -85,B 0,C 180,E1 -29706.081,E2 -29706.081} C_VEL
LIN {X 0,Y 56.154,Z 277.4,A -85,B 0,C 180,E1 -29715.768,E2 -29715.768} C_VEL
LIN {X 0,Y 55.835,Z 276.152,A -85,B 0,C 180,E1 -29720.299,E2 -29720.299} C_VEL
LIN {X 0,Y 55.702,Z 276.42,A -85,B 0,C 180,E1 -29728.883,E2 -29728.883} C_VEL
LIN {X 0,Y 57.661,Z 280.687,A -85,B 0,C 180,E1 -29744.093,E2 -29744.093} C_VEL
LIN {X 0,Y 58.618,Z 281.524,A -85,B 0,C 180,E1 -29747.333,E2 -29747.333} C_VEL
LIN {X 0,Y 60.537,Z 284.884,A -85,B 0,C 180,E1 -29753.236,E2 -29753.236} C_VEL
LIN {X 0,Y 61.444,Z 286.134,A -85,B 0,C 180,E1 -29755.397,E2 -29755.397} C_VEL
LIN {X 0,Y 64.213,Z 290.747,A -85,B 0,C 180,E1 -29761.109,E2 -29761.109} C_VEL
LIN {X 0,Y 64.526,Z 291.304,A -85,B 0,C 180,E1 -29761.681,E2 -29761.681} C_VEL
LIN {X 0,Y 65.603,Z 294.165,A -85,B 0,C 180,E1 -29763.8,E2 -29763.8} C_VEL
LIN {X 0,Y 66.09,Z 297.725,A -85,B 0,C 180,E1 -29765.279,E2 -29765.279} C_VEL
LIN {X 0,Y 66.625,Z 308.072,A -85,B 0,C 180,E1 -29768.406,E2 -29768.406} C_VEL
LIN {X 0,Y 67.156,Z 310.441,A -85,B 0,C 180,E1 -29769.499,E2 -29769.499} C_VEL
LIN {X 0,Y 69.605,Z 318.719,A -85,B 0,C 180,E1 -29773.509,E2 -29773.509} C_VEL
LIN {X 0,Y 64.722,Z 352.528,A -85,B 0,C 180,E1 -29776.386,E2 -29776.386} C_VEL
LIN {X 0,Y 62.113,Z 364.73,A -85,B 0,C 180,E1 -29778.168,E2 -29778.168} C_VEL
LIN {X 0,Y 58.524,Z 377.161,A -85,B 0,C 180,E1 -29780.933,E2 -29780.933} C_VEL
LIN {X 0,Y 54.05,Z 389.274,A -85,B 0,C 180,E1 -29784.873,E2 -29784.873} C_VEL
LIN {X 0,Y 49.45,Z 399.847,A -85,B 0,C 180,E1 -29790.001,E2 -29790.001} C_VEL
LIN {X 0,Y 44.096,Z 410.92,A -85,B 0,C 180,E1 -29798.015,E2 -29798.015} C_VEL
LIN {X 0,Y 39.199,Z 420.88,A -85,B 0,C 180,E1 -29809.026,E2 -29809.026} C_VEL
LIN {X 0,Y 35.861,Z 429.528,A -85,B 0,C 180,E1 -29823.618,E2 -29823.618} C_VEL
LIN {X 0,Y 34.514,Z 436.007,A -85,B 0,C 180,E1 -29838.568,E2 -29838.568} C_VEL
LIN {X 0,Y 35.752,Z 442.412,A -85,B 0,C 180,E1 -29856.854,E2 -29856.854} C_VEL
LIN {X 0,Y 40.658,Z 448,A -85,B 0,C 180,E1 -29873.939,E2 -29873.939} C_VEL
LIN {X 0,Y 49.717,Z 452.856,A -85,B 0,C 180,E1 -29888.342,E2 -29888.342} C_VEL
LIN {X 0,Y 58.569,Z 455.583,A -85,B 0,C 180,E1 -29896.289,E2 -29896.289} C_VEL
LIN {X 0,Y 68.189,Z 457.336,A -85,B 0,C 180,E1 -29901.951,E2 -29901.951} C_VEL
LIN {X 0,Y 69.935,Z 457.603,A -85,B 0,C 180,E1 -29903.704,E2 -29903.704} C_VEL
LIN {X 0,Y 57.459,Z 456.176,A -85,B 0,C 180,E1 -29911.118,E2 -29911.118} C_VEL
LIN {X 0,Y 47.082,Z 453.46,A -85,B 0,C 180,E1 -29921.731,E2 -29921.731} C_VEL
LIN {X 0,Y 39.535,Z 449.367,A -85,B 0,C 180,E1 -29937.774,E2 -29937.774} C_VEL
LIN {X 0,Y 36.758,Z 445.401,A -85,B 0,C 180,E1 -29952.952,E2 -29952.952} C_VEL
LIN {X 0,Y 36.247,Z 442,A -85,B 0,C 180,E1 -29964.436,E2 -29964.436} C_VEL
LIN {X 0,Y 35.938,Z 436.488,A -85,B 0,C 180,E1 -29978.68,E2 -29978.68} C_VEL
LIN {X 0,Y 37.798,Z 428.5,A -85,B 0,C 180,E1 -29994.727,E2 -29994.727} C_VEL
LIN {X 0,Y 41.333,Z 420.179,A -85,B 0,C 180,E1 -30006.515,E2 -30006.515} C_VEL
LIN {X 0,Y 46.309,Z 409.987,A -85,B 0,C 180,E1 -30016.118,E2 -30016.118} C_VEL
LIN {X 0,Y 51.63,Z 398.617,A -85,B 0,C 180,E1 -30023.093,E2 -30023.093} C_VEL
LIN {X 0,Y 56.233,Z 387.507,A -85,B 0,C 180,E1 -30027.513,E2 -30027.513} C_VEL
LIN {X 0,Y 60.396,Z 375.259,A -85,B 0,C 180,E1 -30030.766,E2 -30030.766} C_VEL
LIN {X 0,Y 63.895,Z 361.709,A -85,B 0,C 180,E1 -30033.087,E2 -30033.087} C_VEL
LIN {X 0,Y 66.496,Z 345.038,A -85,B 0,C 180,E1 -30034.861,E2 -30034.861} C_VEL
LIN {X 0,Y 69.33,Z 323.489,A -85,B 0,C 180,E1 -30036.81,E2 -30036.81} C_VEL
LIN {X 0,Y 66.763,Z 310.972,A -85,B 0,C 180,E1 -30041.787,E2 -30041.787} C_VEL
LIN {X 0,Y 64.707,Z 305.076,A -85,B 0,C 180,E1 -30045.451,E2 -30045.451} C_VEL
LIN {X 0,Y 62.341,Z 299.037,A -85,B 0,C 180,E1 -30050.251,E2 -30050.251} C_VEL
LIN {X 0,Y 58.855,Z 291.521,A -85,B 0,C 180,E1 -30058.697,E2 -30058.697} C_VEL
LIN {X 0,Y 56.748,Z 287.133,A -85,B 0,C 180,E1 -30066.219,E2 -30066.219} C_VEL
LIN {X 0,Y 54.77,Z 284.288,A -85,B 0,C 180,E1 -30077.278,E2 -30077.278} C_VEL
LIN {X 0,Y 54.619,Z 283.16,A -85,B 0,C 180,E1 -30080.771,E2 -30080.771} C_VEL
LIN {X 0,Y 54.483,Z 283.437,A -85,B 0,C 180,E1 -30087.617,E2 -30087.617} C_VEL
LIN {X 0,Y 56.47,Z 287.799,A -85,B 0,C 180,E1 -30104.294,E2 -30104.294} C_VEL
LIN {X 0,Y 58.966,Z 292.265,A -85,B 0,C 180,E1 -30112.82,E2 -30112.82} C_VEL
LIN {X 0,Y 61.262,Z 296.563,A -85,B 0,C 180,E1 -30118.457,E2 -30118.457} C_VEL
LIN {X 0,Y 63.172,Z 299.989,A -85,B 0,C 180,E1 -30122.213,E2 -30122.213} C_VEL
LIN {X 0,Y 66.218,Z 307.292,A -85,B 0,C 180,E1 -30127.795,E2 -30127.795} C_VEL
LIN {X 0,Y 67.156,Z 310.441,A -85,B 0,C 180,E1 -30129.499,E2 -30129.499} C_VEL
LIN {X 0,Y 67.509,Z 313.367,A -85,B 0,C 180,E1 -30130.493,E2 -30130.493} C_VEL
LIN {X 0,Y 66.851,Z 317.872,A -85,B 0,C 180,E1 -30130.832,E2 -30130.832} C_VEL
LIN {X 0,Y 63.39,Z 329.24,A -85,B 0,C 180,E1 -30129.895,E2 -30129.895} C_VEL
LIN {X 0,Y 63.03,Z 331.329,A -85,B 0,C 180,E1 -30130.005,E2 -30130.005} C_VEL
LIN {X 0,Y 59.253,Z 355.048,A -85,B 0,C 180,E1 -30132.048,E2 -30132.048} C_VEL
LIN {X 0,Y 55.895,Z 368.866,A -85,B 0,C 180,E1 -30134.217,E2 -30134.217} C_VEL
LIN {X 0,Y 51.26,Z 382.332,A -85,B 0,C 180,E1 -30137.552,E2 -30137.552} C_VEL
LIN {X 0,Y 46.122,Z 394.44,A -85,B 0,C 180,E1 -30142.298,E2 -30142.298} C_VEL
LIN {X 0,Y 40.625,Z 405.3,A -85,B 0,C 180,E1 -30148.978,E2 -30148.978} C_VEL
LIN {X 0,Y 34.919,Z 415.728,A -85,B 0,C 180,E1 -30159.214,E2 -30159.214} C_VEL
LIN {X 0,Y 30.515,Z 424.413,A -85,B 0,C 180,E1 -30172.901,E2 -30172.901} C_VEL
LIN {X 0,Y 27.929,Z 432.05,A -85,B 0,C 180,E1 -30190.989,E2 -30190.989} C_VEL
LIN {X 0,Y 28.109,Z 439.086,A -85,B 0,C 180,E1 -30213.37,E2 -30213.37} C_VEL
LIN {X 0,Y 32.342,Z 445.022,A -85,B 0,C 180,E1 -30233.767,E2 -30233.767} C_VEL
LIN {X 0,Y 40.816,Z 450.363,A -85,B 0,C 180,E1 -30249.919,E2 -30249.919} C_VEL
LIN {X 0,Y 47.654,Z 453.158,A -85,B 0,C 180,E1 -30257.158,E2 -30257.158} C_VEL
LIN {X 0,Y 55.075,Z 455.317,A -85,B 0,C 180,E1 -30262.511,E2 -30262.511} C_VEL
LIN {X 0,Y 54.154,Z 455.231,A -85,B 0,C 180,E1 -30264.72,E2 -30264.72} C_VEL
LIN {X 0,Y 42.737,Z 452.231,A -85,B 0,C 180,E1 -30274.699,E2 -30274.699} C_VEL
LIN {X 0,Y 33.858,Z 447.852,A -85,B 0,C 180,E1 -30291.488,E2 -30291.488} C_VEL
LIN {X 0,Y 29.896,Z 442.531,A -85,B 0,C 180,E1 -30313.707,E2 -30313.707} C_VEL
LIN {X 0,Y 29.214,Z 438.978,A -85,B 0,C 180,E1 -30326.551,E2 -30326.551} C_VEL
LIN {X 0,Y 29.256,Z 433.01,A -85,B 0,C 180,E1 -30343.897,E2 -30343.897} C_VEL
LIN {X 0,Y 32.353,Z 424.2,A -85,B 0,C 180,E1 -30362.888,E2 -30362.888} C_VEL
LIN {X 0,Y 37.565,Z 413.985,A -85,B 0,C 180,E1 -30376.459,E2 -30376.459} C_VEL
LIN {X 0,Y 43.041,Z 403.688,A -85,B 0,C 180,E1 -30384.718,E2 -30384.718} C_VEL
LIN {X 0,Y 48.475,Z 392.293,A -85,B 0,C 180,E1 -30390.433,E2 -30390.433} C_VEL
LIN {X 0,Y 53.582,Z 379.528,A -85,B 0,C 180,E1 -30394.374,E2 -30394.374} C_VEL
LIN {X 0,Y 57.509,Z 366.586,A -85,B 0,C 180,E1 -30396.965,E2 -30396.965} C_VEL
LIN {X 0,Y 60.233,Z 353.688,A -85,B 0,C 180,E1 -30398.557,E2 -30398.557} C_VEL
LIN {X 0,Y 64.341,Z 325.042,A -85,B 0,C 180,E1 -30401.076,E2 -30401.076} C_VEL
LIN {X 0,Y 62.349,Z 313.788,A -85,B 0,C 180,E1 -30406.139,E2 -30406.139} C_VEL
LIN {X 0,Y 59.65,Z 305.667,A -85,B 0,C 180,E1 -30412.328,E2 -30412.328} C_VEL
LIN {X 0,Y 57.603,Z 300.63,A -85,B 0,C 180,E1 -30417.783,E2 -30417.783} C_VEL
LIN {X 0,Y 56.082,Z 296.654,A -85,B 0,C 180,E1 -30423.144,E2 -30423.144} C_VEL
LIN {X 0,Y 54.83,Z 293.641,A -85,B 0,C 180,E1 -30428.917,E2 -30428.917} C_VEL
LIN {X 0,Y 53.395,Z 290.776,A -85,B 0,C 180,E1 -30439.967,E2 -30439.967} C_VEL
LIN {X 0,Y 53.341,Z 290.152,A -85,B 0,C 180,E1 -30442.754,E2 -30442.754} C_VEL
LIN {X 0,Y 53.266,Z 290.6,A -85,B 0,C 180,E1 -30447.01,E2 -30447.01} C_VEL
LIN {X 0,Y 54.858,Z 294.794,A -85,B 0,C 180,E1 -30463.026,E2 -30463.026} C_VEL
LIN {X 0,Y 56.761,Z 298.72,A -85,B 0,C 180,E1 -30470.523,E2 -30470.523} C_VEL
LIN {X 0,Y 59.563,Z 304.474,A -85,B 0,C 180,E1 -30478.197,E2 -30478.197} C_VEL
LIN {X 0,Y 62.229,Z 311.39,A -85,B 0,C 180,E1 -30484.025,E2 -30484.025} C_VEL
LIN {X 0,Y 64.579,Z 320.337,A -85,B 0,C 180,E1 -30489.074,E2 -30489.074} C_VEL
LIN {X 0,Y 63.03,Z 331.329,A -85,B 0,C 180,E1 -30490.005,E2 -30490.005} C_VEL
LIN {X 0,Y 61.865,Z 337.099,A -85,B 0,C 180,E1 -30490.104,E2 -30490.104} C_VEL
LIN {X 0,Y 58.662,Z 346.359,A -85,B 0,C 180,E1 -30488.822,E2 -30488.822} C_VEL
LIN {X 0,Y 55.075,Z 355.532,A -85,B 0,C 180,E1 -30487.331,E2 -30487.331} C_VEL
LIN {X 0,Y 53.238,Z 361.181,A -85,B 0,C 180,E1 -30487.391,E2 -30487.391} C_VEL
LIN {X 0,Y 49.641,Z 373.207,A -85,B 0,C 180,E1 -30489.437,E2 -30489.437} C_VEL
LIN {X 0,Y 44.653,Z 385.833,A -85,B 0,C 180,E1 -30492.767,E2 -30492.767} C_VEL
LIN {X 0,Y 39.378,Z 396.752,A -85,B 0,C 180,E1 -30497.417,E2 -30497.417} C_VEL
LIN {X 0,Y 33.063,Z 407.92,A -85,B 0,C 180,E1 -30505.142,E2 -30505.142} C_VEL
LIN {X 0,Y 26.948,Z 417.902,A -85,B 0,C 180,E1 -30517.314,E2 -30517.314} C_VEL
LIN {X 0,Y 22.123,Z 427.203,A -85,B 0,C 180,E1 -30538.219,E2 -30538.219} C_VEL
LIN {X 0,Y 20.584,Z 434.199,A -85,B 0,C 180,E1 -30563.317,E2 -30563.317} C_VEL
LIN {X 0,Y 23.8,Z 441.144,A -85,B 0,C 180,E1 -30592.165,E2 -30592.165} C_VEL
LIN {X 0,Y 32.185,Z 447.367,A -85,B 0,C 180,E1 -30612.617,E2 -30612.617} C_VEL
LIN {X 0,Y 41.055,Z 451.429,A -85,B 0,C 180,E1 -30622.482,E2 -30622.482} C_VEL
LIN {X 0,Y 39.182,Z 450.875,A -85,B 0,C 180,E1 -30626.266,E2 -30626.266} C_VEL
LIN {X 0,Y 28.772,Z 446.195,A -85,B 0,C 180,E1 -30642.884,E2 -30642.884} C_VEL
LIN {X 0,Y 23.631,Z 441.151,A -85,B 0,C 180,E1 -30666.481,E2 -30666.481} C_VEL
LIN {X 0,Y 22.597,Z 437.959,A -85,B 0,C 180,E1 -30681.053,E2 -30681.053} C_VEL
LIN {X 0,Y 22.331,Z 431.557,A -85,B 0,C 180,E1 -30704.794,E2 -30704.794} C_VEL
LIN {X 0,Y 25.835,Z 422.851,A -85,B 0,C 180,E1 -30727.733,E2 -30727.733} C_VEL
LIN {X 0,Y 31.871,Z 412.468,A -85,B 0,C 180,E1 -30743.06,E2 -30743.06} C_VEL
LIN {X 0,Y 37.99,Z 401.989,A -85,B 0,C 180,E1 -30751.476,E2 -30751.476} C_VEL
LIN {X 0,Y 43.916,Z 390.273,A -85,B 0,C 180,E1 -30756.938,E2 -30756.938} C_VEL
LIN {X 0,Y 48.98,Z 378.215,A -85,B 0,C 180,E1 -30760.307,E2 -30760.307} C_VEL
LIN {X 0,Y 52.926,Z 365.758,A -85,B 0,C 180,E1 -30762.509,E2 -30762.509} C_VEL
LIN {X 0,Y 55.664,Z 353.283,A -85,B 0,C 180,E1 -30763.919,E2 -30763.919} C_VEL
LIN {X 0,Y 59.717,Z 326.343,A -85,B 0,C 180,E1 -30766.168,E2 -30766.168} C_VEL
LIN {X 0,Y 58.347,Z 317.049,A -85,B 0,C 180,E1 -30770.838,E2 -30770.838} C_VEL
LIN {X 0,Y 56.179,Z 309.594,A -85,B 0,C 180,E1 -30777.271,E2 -30777.271} C_VEL
LIN {X 0,Y 54.098,Z 302.954,A -85,B 0,C 180,E1 -30785.781,E2 -30785.781} C_VEL
LIN {X 0,Y 53.053,Z 300.221,A -85,B 0,C 180,E1 -30791.491,E2 -30791.491} C_VEL
LIN {X 0,Y 52.13,Z 297.195,A -85,B 0,C 180,E1 -30803.854,E2 -30803.854} C_VEL
LIN {X 0,Y 53.168,Z 301.583,A -85,B 0,C 180,E1 -30821.114,E2 -30821.114} C_VEL
LIN {X 0,Y 54.623,Z 305.066,A -85,B 0,C 180,E1 -30827.898,E2 -30827.898} C_VEL
LIN {X 0,Y 56.775,Z 310.419,A -85,B 0,C 180,E1 -30835.245,E2 -30835.245} C_VEL
LIN {X 0,Y 58.565,Z 316.05,A -85,B 0,C 180,E1 -30840.244,E2 -30840.244} C_VEL
LIN {X 0,Y 59.998,Z 322.449,A -85,B 0,C 180,E1 -30844.129,E2 -30844.129} C_VEL
LIN {X 0,Y 54.663,Z 354.975,A -85,B 0,C 180,E1 -30846.609,E2 -30846.609} C_VEL
LIN {X 0,Y 53.238,Z 361.181,A -85,B 0,C 180,E1 -30847.391,E2 -30847.391} C_VEL
LIN {X 0,Y 51.203,Z 366.738,A -85,B 0,C 180,E1 -30847.53,E2 -30847.53} C_VEL
LIN {X 0,Y 46.469,Z 375.423,A -85,B 0,C 180,E1 -30846.453,E2 -30846.453} C_VEL
LIN {X 0,Y 41.27,Z 383.908,A -85,B 0,C 180,E1 -30845.555,E2 -30845.555} C_VEL
LIN {X 0,Y 38.48,Z 389.075,A -85,B 0,C 180,E1 -30846.449,E2 -30846.449} C_VEL
LIN {X 0,Y 32.477,Z 399.991,A -85,B 0,C 180,E1 -30851.062,E2 -30851.062} C_VEL
LIN {X 0,Y 25.202,Z 411.242,A -85,B 0,C 180,E1 -30860.042,E2 -30860.042} C_VEL
LIN {X 0,Y 18.101,Z 421.31,A -85,B 0,C 180,E1 -30877.245,E2 -30877.245} C_VEL
LIN {X 0,Y 14.134,Z 428.968,A -85,B 0,C 180,E1 -30905.863,E2 -30905.863} C_VEL
LIN {X 0,Y 14.686,Z 435.541,A -85,B 0,C 180,E1 -30943.148,E2 -30943.148} C_VEL
LIN {X 0,Y 21.669,Z 442.364,A -85,B 0,C 180,E1 -30973.369,E2 -30973.369} C_VEL
LIN {X 0,Y 28.046,Z 446.081,A -85,B 0,C 180,E1 -30983.365,E2 -30983.365} C_VEL
LIN {X 0,Y 26.061,Z 445.203,A -85,B 0,C 180,E1 -30988.349,E2 -30988.349} C_VEL
LIN {X 0,Y 18.023,Z 439.606,A -85,B 0,C 180,E1 -31014.616,E2 -31014.616} C_VEL
LIN {X 0,Y 16.305,Z 436.817,A -85,B 0,C 180,E1 -31031.139,E2 -31031.139} C_VEL
LIN {X 0,Y 15.232,Z 430.917,A -85,B 0,C 180,E1 -31062.358,E2 -31062.358} C_VEL
LIN {X 0,Y 19.626,Z 421.491,A -85,B 0,C 180,E1 -31095.733,E2 -31095.733} C_VEL
LIN {X 0,Y 26.781,Z 410.907,A -85,B 0,C 180,E1 -31112.323,E2 -31112.323} C_VEL
LIN {X 0,Y 33.634,Z 400.091,A -85,B 0,C 180,E1 -31120.082,E2 -31120.082} C_VEL
LIN {X 0,Y 40.057,Z 388.042,A -85,B 0,C 180,E1 -31124.763,E2 -31124.763} C_VEL
LIN {X 0,Y 45.44,Z 375.321,A -85,B 0,C 180,E1 -31127.477,E2 -31127.477} C_VEL
LIN {X 0,Y 49.619,Z 361.862,A -85,B 0,C 180,E1 -31129.268,E2 -31129.268} C_VEL
LIN {X 0,Y 52.428,Z 347.655,A -85,B 0,C 180,E1 -31130.464,E2 -31130.464} C_VEL
LIN {X 0,Y 55.538,Z 327.721,A -85,B 0,C 180,E1 -31131.936,E2 -31131.936} C_VEL
LIN {X 0,Y 54.792,Z 320.844,A -85,B 0,C 180,E1 -31135.757,E2 -31135.757} C_VEL
LIN {X 0,Y 53.294,Z 314.159,A -85,B 0,C 180,E1 -31142.16,E2 -31142.16} C_VEL
LIN {X 0,Y 51.958,Z 308.695,A -85,B 0,C 180,E1 -31149.877,E2 -31149.877} C_VEL
LIN {X 0,Y 51.419,Z 306.776,A -85,B 0,C 180,E1 -31154.091,E2 -31154.091} C_VEL
LIN {X 0,Y 50.902,Z 304.651,A -85,B 0,C 180,E1 -31162.793,E2 -31162.793} C_VEL
LIN {X 0,Y 50.853,Z 304.754,A -85,B 0,C 180,E1 -31165.322,E2 -31165.322} C_VEL
LIN {X 0,Y 51.483,Z 308.159,A -85,B 0,C 180,E1 -31178.603,E2 -31178.603} C_VEL
LIN {X 0,Y 52.557,Z 311.383,A -85,B 0,C 180,E1 -31185.117,E2 -31185.117} C_VEL
LIN {X 0,Y 54.035,Z 315.919,A -85,B 0,C 180,E1 -31191.533,E2 -31191.533} C_VEL
LIN {X 0,Y 55.122,Z 320.393,A -85,B 0,C 180,E1 -31195.729,E2 -31195.729} C_VEL
LIN {X 0,Y 55.821,Z 324.185,A -85,B 0,C 180,E1 -31198.383,E2 -31198.383} C_VEL
LIN {X 0,Y 50.493,Z 355.122,A -85,B 0,C 180,E1 -31200.289,E2 -31200.289} C_VEL
LIN {X 0,Y 46.828,Z 368.79,A -85,B 0,C 180,E1 -31201.939,E2 -31201.939} C_VEL
LIN {X 0,Y 42.286,Z 380.822,A -85,B 0,C 180,E1 -31204.137,E2 -31204.137} C_VEL
LIN {X 0,Y 38.48,Z 389.075,A -85,B 0,C 180,E1 -31206.449,E2 -31206.449} C_VEL
LIN {X 0,Y 35.505,Z 394.119,A -85,B 0,C 180,E1 -31207.514,E2 -31207.514} C_VEL
LIN {X 0,Y 29.156,Z 401.724,A -85,B 0,C 180,E1 -31207.146,E2 -31207.146} C_VEL
LIN {X 0,Y 22.228,Z 408.963,A -85,B 0,C 180,E1 -31206.686,E2 -31206.686} C_VEL
LIN {X 0,Y 18.313,Z 413.363,A -85,B 0,C 180,E1 -31209.172,E2 -31209.172} C_VEL
LIN {X 0,Y 9.832,Z 423.647,A -85,B 0,C 180,E1 -31233.392,E2 -31233.392} C_VEL
LIN {X 0,Y 7.314,Z 431.807,A -85,B 0,C 180,E1 -31303.931,E2 -31303.931} C_VEL
LIN {X 0,Y 15.595,Z 439.201,A -85,B 0,C 180,E1 -31346.797,E2 -31346.797} C_VEL
LIN {X 0,Y 11.055,Z 435.579,A -85,B 0,C 180,E1 -31370.527,E2 -31370.527} C_VEL
LIN {X 0,Y 8.622,Z 432.041,A -85,B 0,C 180,E1 -31398.239,E2 -31398.239} C_VEL
LIN {X 0,Y 11.447,Z 423.369,A -85,B 0,C 180,E1 -31460.229,E2 -31460.229} C_VEL
LIN {X 0,Y 18.661,Z 414.448,A -85,B 0,C 180,E1 -31480.284,E2 -31480.284} C_VEL
LIN {X 0,Y 26.87,Z 403.439,A -85,B 0,C 180,E1 -31488.725,E2 -31488.725} C_VEL
LIN {X 0,Y 33.658,Z 392.377,A -85,B 0,C 180,E1 -31492.608,E2 -31492.608} C_VEL
LIN {X 0,Y 40.124,Z 379.021,A -85,B 0,C 180,E1 -31494.923,E2 -31494.923} C_VEL
LIN {X 0,Y 44.891,Z 365.712,A -85,B 0,C 180,E1 -31496.315,E2 -31496.315} C_VEL
LIN {X 0,Y 47.964,Z 353.154,A -85,B 0,C 180,E1 -31497.13,E2 -31497.13} C_VEL
LIN {X 0,Y 51.962,Z 329.472,A -85,B 0,C 180,E1 -31498.363,E2 -31498.363} C_VEL
LIN {X 0,Y 51.647,Z 324.44,A -85,B 0,C 180,E1 -31501.539,E2 -31501.539} C_VEL
LIN {X 0,Y 50.794,Z 318.826,A -85,B 0,C 180,E1 -31507.502,E2 -31507.502} C_VEL
LIN {X 0,Y 50.094,Z 314.439,A -85,B 0,C 180,E1 -31514.159,E2 -31514.159} C_VEL
LIN {X 0,Y 49.872,Z 313.313,A -85,B 0,C 180,E1 -31517.08,E2 -31517.08} C_VEL
LIN {X 0,Y 49.676,Z 311.916,A -85,B 0,C 180,E1 -31522.962,E2 -31522.962} C_VEL
LIN {X 0,Y 49.619,Z 312.137,A -85,B 0,C 180,E1 -31525.944,E2 -31525.944} C_VEL
LIN {X 0,Y 49.902,Z 314.745,A -85,B 0,C 180,E1 -31535.972,E2 -31535.972} C_VEL
LIN {X 0,Y 50.63,Z 317.804,A -85,B 0,C 180,E1 -31542.31,E2 -31542.31} C_VEL
LIN {X 0,Y 51.545,Z 321.641,A -85,B 0,C 180,E1 -31547.649,E2 -31547.649} C_VEL
LIN {X 0,Y 52.092,Z 325.023,A -85,B 0,C 180,E1 -31550.869,E2 -31550.869} C_VEL
LIN {X 0,Y 52.223,Z 326.068,A -85,B 0,C 180,E1 -31551.69,E2 -31551.69} C_VEL
LIN {X 0,Y 47.213,Z 354.619,A -85,B 0,C 180,E1 -31552.947,E2 -31552.947} C_VEL
LIN {X 0,Y 43.41,Z 368.418,A -85,B 0,C 180,E1 -31554.041,E2 -31554.041} C_VEL
LIN {X 0,Y 38.388,Z 381.182,A -85,B 0,C 180,E1 -31555.562,E2 -31555.562} C_VEL
LIN {X 0,Y 32.209,Z 393.273,A -85,B 0,C 180,E1 -31558.153,E2 -31558.153} C_VEL
LIN {X 0,Y 24.495,Z 405.287,A -85,B 0,C 180,E1 -31562.823,E2 -31562.823} C_VEL
LIN {X 0,Y 18.313,Z 413.363,A -85,B 0,C 180,E1 -31569.172,E2 -31569.172} C_VEL
LIN {X 0,Y 15.57,Z 416.181,A -85,B 0,C 180,E1 -31570.831,E2 -31570.831} C_VEL
LIN {X 0,Y 10.18,Z 420.119,A -85,B 0,C 180,E1 -31567.756,E2 -31567.756} C_VEL
LIN {X 0,Y 4.63,Z 423.801,A -85,B 0,C 180,E1 -31556.958,E2 -31556.958} C_VEL
LIN {X 0,Y 1.463,Z 426.236,A -85,B 0,C 180,E1 -31547.167,E2 -31547.167} C_VEL
LIN {X 0,Y 0.123,Z 427.522,A -85,B 0,C 180,E1 -31409.714,E2 -31409.714} C_VEL
LIN {X 0,Y 1.398,Z 428.031,A -85,B 0,C 180,E1 -31409.975,E2 -31409.975} C_VEL
LIN {X 0,Y 9.975,Z 419.056,A -85,B 0,C 180,E1 -31498.038,E2 -31498.038} C_VEL
LIN {X 0,Y 18.46,Z 409.575,A -85,B 0,C 180,E1 -31502.233,E2 -31502.233} C_VEL
LIN {X 0,Y 26.403,Z 398.755,A -85,B 0,C 180,E1 -31503.58,E2 -31503.58} C_VEL
LIN {X 0,Y 33.478,Z 386.631,A -85,B 0,C 180,E1 -31504.426,E2 -31504.426} C_VEL
LIN {X 0,Y 39.221,Z 373.805,A -85,B 0,C 180,E1 -31504.709,E2 -31504.709} C_VEL
LIN {X 0,Y 43.495,Z 360.684,A -85,B 0,C 180,E1 -31505.036,E2 -31505.036} C_VEL
LIN {X 0,Y 46.549,Z 345.908,A -85,B 0,C 180,E1 -31505.411,E2 -31505.411} C_VEL
LIN {X 0,Y 49.121,Z 330.665,A -85,B 0,C 180,E1 -31505.97,E2 -31505.97} C_VEL
LIN {X 0,Y 49.026,Z 328.073,A -85,B 0,C 180,E1 -31507.98,E2 -31507.98} C_VEL
LIN {X 0,Y 48.683,Z 323.677,A -85,B 0,C 180,E1 -31513.073,E2 -31513.073} C_VEL
LIN {X 0,Y 48.526,Z 320.414,A -85,B 0,C 180,E1 -31518.307,E2 -31518.307} C_VEL
LIN {X 0,Y 48.439,Z 319.501,A -85,B 0,C 180,E1 -31521.657,E2 -31521.657} C_VEL
LIN {X 0,Y 48.379,Z 319.482,A -85,B 0,C 180,E1 -31526.246,E2 -31526.246} C_VEL
LIN {X 0,Y 48.461,Z 321.481,A -85,B 0,C 180,E1 -31533.711,E2 -31533.711} C_VEL
LIN {X 0,Y 48.871,Z 324.755,A -85,B 0,C 180,E1 -31539.939,E2 -31539.939} C_VEL
LIN {X 0,Y 49.314,Z 328.059,A -85,B 0,C 180,E1 -31544.199,E2 -31544.199} C_VEL
LIN {X 0,Y 45.483,Z 350.055,A -85,B 0,C 180,E1 -31544.645,E2 -31544.645} C_VEL
LIN {X 0,Y 42.141,Z 363.811,A -85,B 0,C 180,E1 -31544.957,E2 -31544.957} C_VEL
LIN {X 0,Y 37.921,Z 375.764,A -85,B 0,C 180,E1 -31545.274,E2 -31545.274} C_VEL
LIN {X 0,Y 31.602,Z 389.053,A -85,B 0,C 180,E1 -31545.761,E2 -31545.761} C_VEL
LIN {X 0,Y 24.207,Z 401.129,A -85,B 0,C 180,E1 -31546.466,E2 -31546.466} C_VEL
LIN {X 0,Y 15.607,Z 412.216,A -85,B 0,C 180,E1 -31547.173,E2 -31547.173} C_VEL
LIN {X 0,Y 5.827,Z 422.45,A -85,B 0,C 180,E1 -31548.885,E2 -31548.885} C_VEL
LIN {X 0,Y 1.463,Z 426.236,A -85,B 0,C 180,E1 -31547.167,E2 -31547.167} C_VEL
LIN {X 0,Y 1.899,Z 425.799,A -85,B 0,C 180,E1 -31518.767,E2 -31518.767} C_VEL
LIN {X 0,Y 3.074,Z 424.761,A -85,B 0,C 180,E1 -31512.872,E2 -31512.872} C_VEL
LIN {X 0,Y 9.024,Z 418.811,A -85,B 0,C 180,E1 -31520.11,E2 -31520.11} C_VEL
LIN {X 0,Y 17.149,Z 409.154,A -85,B 0,C 180,E1 -31526.455,E2 -31526.455} C_VEL
LIN {X 0,Y 21.533,Z 403.134,A -85,B 0,C 180,E1 -31528.631,E2 -31528.631} C_VEL
LIN {X 0,Y 25.612,Z 396.92,A -85,B 0,C 180,E1 -31530.745,E2 -31530.745} C_VEL
LIN {X 0,Y 32.077,Z 385.235,A -85,B 0,C 180,E1 -31533.364,E2 -31533.364} C_VEL
LIN {X 0,Y 37.485,Z 372.689,A -85,B 0,C 180,E1 -31534.754,E2 -31534.754} C_VEL
LIN {X 0,Y 41.75,Z 359.291,A -85,B 0,C 180,E1 -31535.552,E2 -31535.552} C_VEL
LIN {X 0,Y 45.257,Z 341.845,A -85,B 0,C 180,E1 -31536.052,E2 -31536.052} C_VEL
LIN {X 0,Y 47.113,Z 331.165,A -85,B 0,C 180,E1 -31536.196,E2 -31536.196} C_VEL
LIN {X 0,Y 47.091,Z 328.332,A -85,B 0,C 180,E1 -31531.491,E2 -31531.491} C_VEL
LIN {X 0,Y 47.139,Z 326.837,A -85,B 0,C 180,E1 -31526.565,E2 -31526.565} C_VEL
LIN {X 0,Y 47.193,Z 326.414,A -85,B 0,C 180,E1 -31524.245,E2 -31524.245} C_VEL
LIN {X 0,Y 47.183,Z 326.926,A -85,B 0,C 180,E1 -31521.544,E2 -31521.544} C_VEL
LIN {X 0,Y 47.009,Z 331.235,A -85,B 0,C 180,E1 -31515.444,E2 -31515.444} C_VEL
LIN {X 0,Y 46.983,Z 332.714,A -85,B 0,C 180,E1 -31513.898,E2 -31513.898} C_VEL
LIN {X 0,Y 42.4,Z 357.475,A -85,B 0,C 180,E1 -31514.071,E2 -31514.071} C_VEL
LIN {X 0,Y 38.601,Z 370.325,A -85,B 0,C 180,E1 -31514.735,E2 -31514.735} C_VEL
LIN {X 0,Y 33.796,Z 382.097,A -85,B 0,C 180,E1 -31515.917,E2 -31515.917} C_VEL
LIN {X 0,Y 27.694,Z 393.684,A -85,B 0,C 180,E1 -31517.914,E2 -31517.914} C_VEL
LIN {X 0,Y 20.951,Z 404.06,A -85,B 0,C 180,E1 -31521.404,E2 -31521.404} C_VEL
LIN {X 0,Y 19.765,Z 405.663,A -85,B 0,C 180,E1 -31526.554,E2 -31526.554} C_VEL
LIN {X 0,Y 25.612,Z 396.92,A -85,B 0,C 180,E1 -31530.745,E2 -31530.745} C_VEL
LIN {X 0,Y 30.19,Z 388.92,A -85,B 0,C 180,E1 -31531.42,E2 -31531.42} C_VEL
LIN {X 0,Y 34.09,Z 380.568,A -85,B 0,C 180,E1 -31529.777,E2 -31529.777} C_VEL
LIN {X 0,Y 38.386,Z 368.992,A -85,B 0,C 180,E1 -31526.595,E2 -31526.595} C_VEL
LIN {X 0,Y 41.752,Z 356.95,A -85,B 0,C 180,E1 -31524.037,E2 -31524.037} C_VEL
LIN {X 0,Y 43.042,Z 350.793,A -85,B 0,C 180,E1 -31523.374,E2 -31523.374} C_VEL
LIN {X 0,Y 45.752,Z 335.068,A -85,B 0,C 180,E1 -31522.848,E2 -31522.848} C_VEL
LIN {X 0,Y 45.945,Z 333.765,A -85,B 0,C 180,E1 -31524.948,E2 -31524.948} C_VEL
LIN {X 0,Y 45.865,Z 334.484,A -85,B 0,C 180,E1 -31527.364,E2 -31527.364} C_VEL
LIN {X 0,Y 41.635,Z 357.445,A -85,B 0,C 180,E1 -31525.943,E2 -31525.943} C_VEL
LIN {X 0,Y 40.739,Z 361.057,A -85,B 0,C 180,E1 -31525.545,E2 -31525.545} C_VEL
LIN {X 0,Y 40.715,Z 361.159,A -85,B 0,C 180,E1 -31524.243,E2 -31524.243} C_VEL
LIN {X 0,Y 43.042,Z 350.793,A -85,B 0,C 180,E1 -31523.374,E2 -31523.374} C_VEL
LIN {X 0,Y 46.96,Z 351.175,A -85,B 0,C 180,E1 -31522.61,E2 -31522.61} C_VEL
LIN {X 0,Y 46.96,Z 600,A -85,B 0,C 180,E1 -31522.61,E2 -31522.61} C_VEL
LIN {X 0,Y 46.96,Z 600,A -85,B 0,C 180,E1 -31522.61,E2 -31522.61}

QRS_NEXT_CUT()

QRS_NEXT()
QRS_HOME()

END
